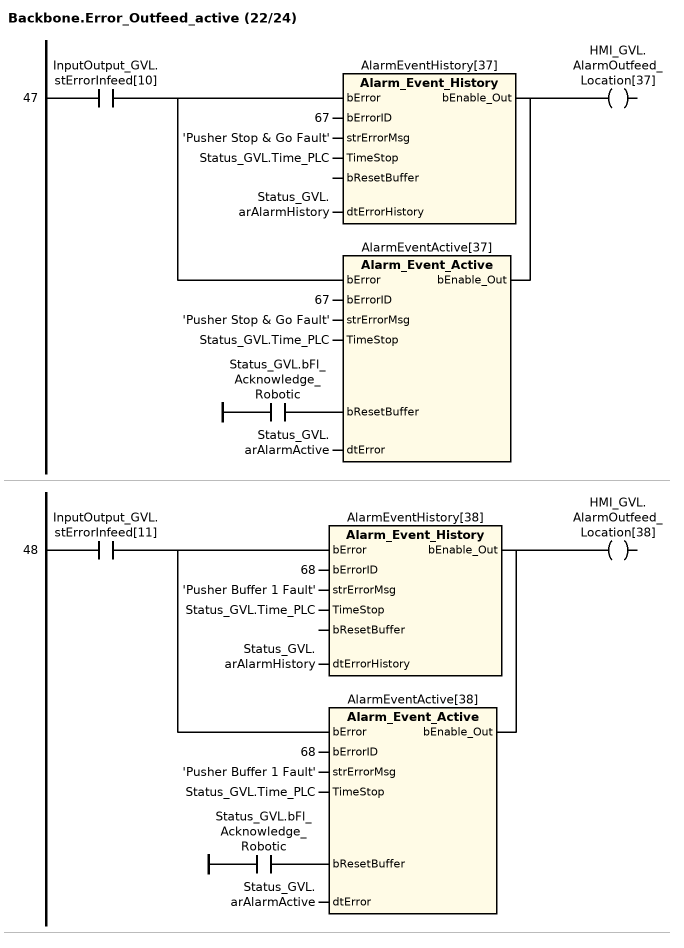
// NETWORK 47
AlarmEventHistory[37](
    bError := InputOutput_GVL.stErrorInfeed[10],
    bErrorID := 67,
    strErrorMsg := 'Pusher Stop & Go Fault',
    TimeStop := Status_GVL.Time_PLC,
    dtErrorHistory := Status_GVL.arAlarmHistory); // Alarm_Event_History
AlarmEventActive[37](
    bError := InputOutput_GVL.stErrorInfeed[10],
    bErrorID := 67,
    strErrorMsg := 'Pusher Stop & Go Fault',
    TimeStop := Status_GVL.Time_PLC,
    bResetBuffer := Status_GVL.bFl_Acknowledge_Robotic,
    dtError := Status_GVL.arAlarmActive); // Alarm_Event_Active
HMI_GVL.AlarmOutfeed_Location[37] := AlarmEventHistory[37].bEnable_Out OR AlarmEventActive[37].bEnable_Out;

// NETWORK 48
AlarmEventHistory[38](
    bError := InputOutput_GVL.stErrorInfeed[11],
    bErrorID := 68,
    strErrorMsg := 'Pusher Buffer 1 Fault',
    TimeStop := Status_GVL.Time_PLC,
    dtErrorHistory := Status_GVL.arAlarmHistory); // Alarm_Event_History
AlarmEventActive[38](
    bError := InputOutput_GVL.stErrorInfeed[11],
    bErrorID := 68,
    strErrorMsg := 'Pusher Buffer 1 Fault',
    TimeStop := Status_GVL.Time_PLC,
    bResetBuffer := Status_GVL.bFl_Acknowledge_Robotic,
    dtError := Status_GVL.arAlarmActive); // Alarm_Event_Active
HMI_GVL.AlarmOutfeed_Location[38] := AlarmEventHistory[38].bEnable_Out OR AlarmEventActive[38].bEnable_Out;

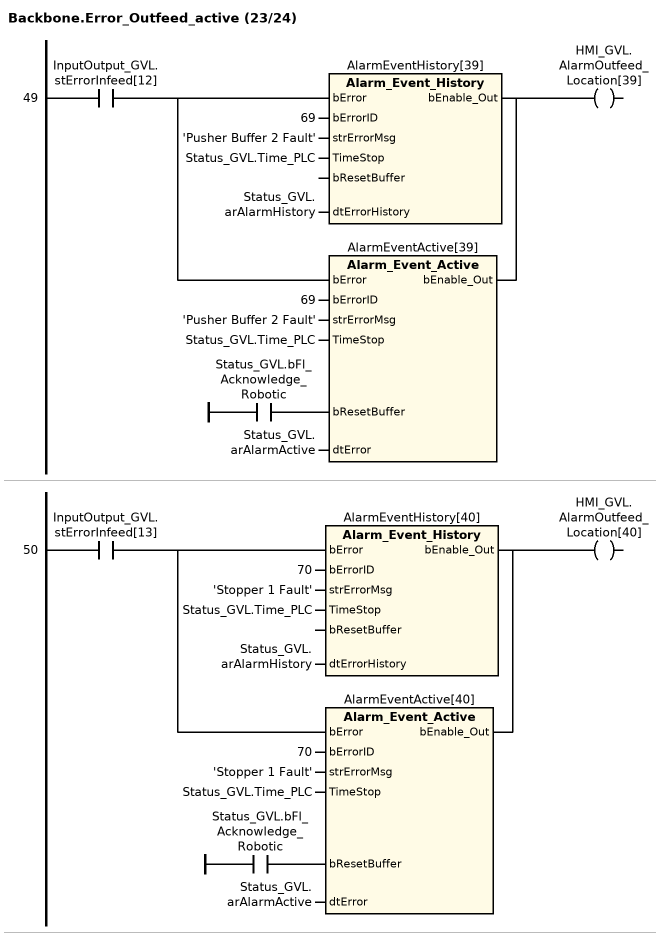
// NETWORK 49
AlarmEventHistory[39](
    bError := InputOutput_GVL.stErrorInfeed[12],
    bErrorID := 69,
    strErrorMsg := 'Pusher Buffer 2 Fault',
    TimeStop := Status_GVL.Time_PLC,
    dtErrorHistory := Status_GVL.arAlarmHistory); // Alarm_Event_History
AlarmEventActive[39](
    bError := InputOutput_GVL.stErrorInfeed[12],
    bErrorID := 69,
    strErrorMsg := 'Pusher Buffer 2 Fault',
    TimeStop := Status_GVL.Time_PLC,
    bResetBuffer := Status_GVL.bFl_Acknowledge_Robotic,
    dtError := Status_GVL.arAlarmActive); // Alarm_Event_Active
HMI_GVL.AlarmOutfeed_Location[39] := AlarmEventHistory[39].bEnable_Out OR AlarmEventActive[39].bEnable_Out;

// NETWORK 50
AlarmEventHistory[40](
    bError := InputOutput_GVL.stErrorInfeed[13],
    bErrorID := 70,
    strErrorMsg := 'Stopper 1 Fault',
    TimeStop := Status_GVL.Time_PLC,
    dtErrorHistory := Status_GVL.arAlarmHistory); // Alarm_Event_History
AlarmEventActive[40](
    bError := InputOutput_GVL.stErrorInfeed[13],
    bErrorID := 70,
    strErrorMsg := 'Stopper 1 Fault',
    TimeStop := Status_GVL.Time_PLC,
    bResetBuffer := Status_GVL.bFl_Acknowledge_Robotic,
    dtError := Status_GVL.arAlarmActive); // Alarm_Event_Active
HMI_GVL.AlarmOutfeed_Location[40] := AlarmEventHistory[40].bEnable_Out OR AlarmEventActive[40].bEnable_Out;

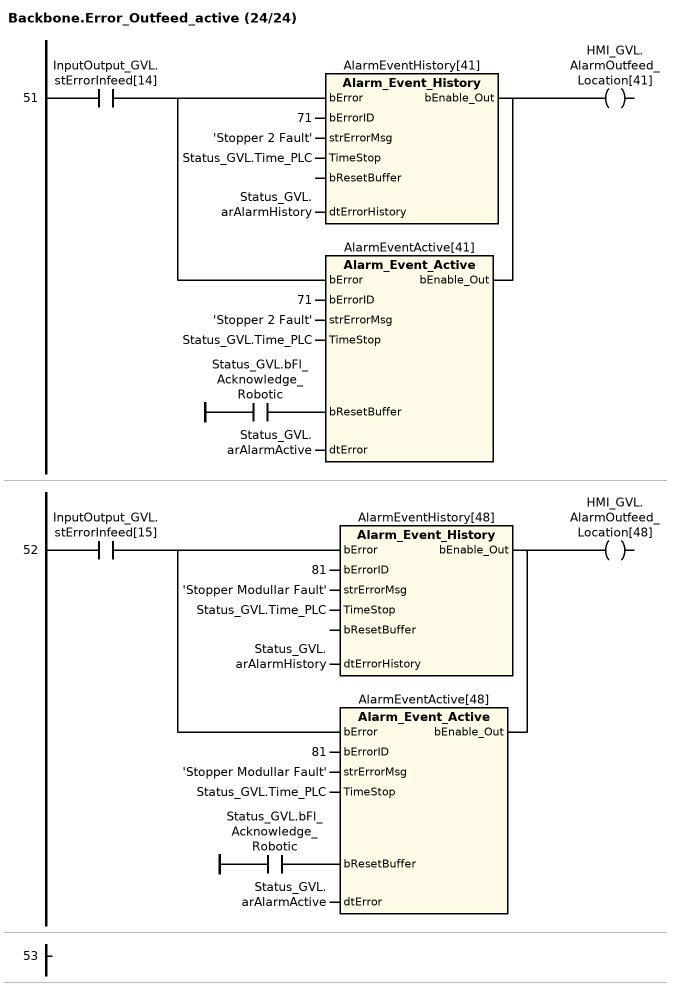
// NETWORK 51
AlarmEventHistory[41](
    bError := InputOutput_GVL.stErrorInfeed[14],
    bErrorID := 71,
    strErrorMsg := 'Stopper 2 Fault',
    TimeStop := Status_GVL.Time_PLC,
    dtErrorHistory := Status_GVL.arAlarmHistory); // Alarm_Event_History
AlarmEventActive[41](
    bError := InputOutput_GVL.stErrorInfeed[14],
    bErrorID := 71,
    strErrorMsg := 'Stopper 2 Fault',
    TimeStop := Status_GVL.Time_PLC,
    bResetBuffer := Status_GVL.bFl_Acknowledge_Robotic,
    dtError := Status_GVL.arAlarmActive); // Alarm_Event_Active
HMI_GVL.AlarmOutfeed_Location[41] := AlarmEventHistory[41].bEnable_Out OR AlarmEventActive[41].bEnable_Out;

// NETWORK 52
AlarmEventHistory[48](
    bError := InputOutput_GVL.stErrorInfeed[15],
    bErrorID := 81,
    strErrorMsg := 'Stopper Modullar Fault',
    TimeStop := Status_GVL.Time_PLC,
    dtErrorHistory := Status_GVL.arAlarmHistory); // Alarm_Event_History
AlarmEventActive[48](
    bError := InputOutput_GVL.stErrorInfeed[15],
    bErrorID := 81,
    strErrorMsg := 'Stopper Modullar Fault',
    TimeStop := Status_GVL.Time_PLC,
    bResetBuffer := Status_GVL.bFl_Acknowledge_Robotic,
    dtError := Status_GVL.arAlarmActive); // Alarm_Event_Active
HMI_GVL.AlarmOutfeed_Location[48] := AlarmEventHistory[48].bEnable_Out OR AlarmEventActive[48].bEnable_Out;

// NETWORK 53
END_ACTION

ACTION FGHS_DataCollect_active:
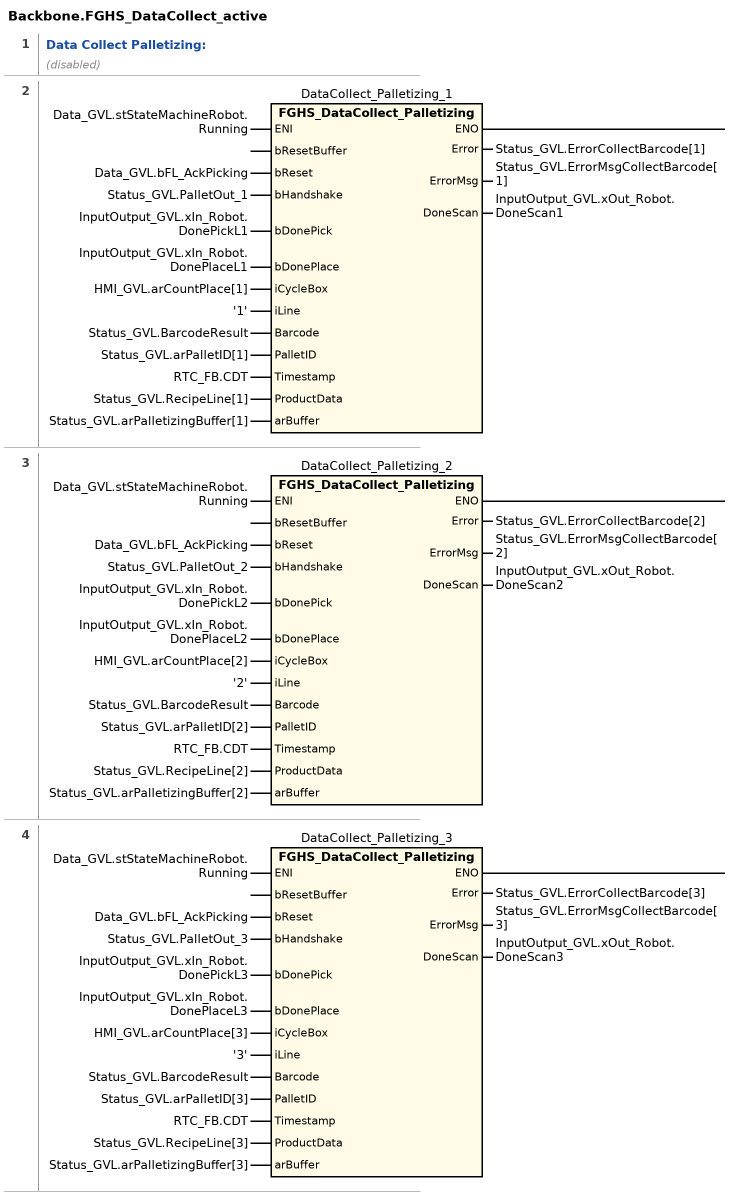
// NETWORK 1 (disabled)
// label: Data Collect Palletizing

// NETWORK 2
DataCollect_Palletizing_1(
    ENI := Data_GVL.stStateMachineRobot.Running,
    bReset := Data_GVL.bFL_AckPicking,
    bHandshake := Status_GVL.PalletOut_1,
    bDonePick := InputOutput_GVL.xIn_Robot.DonePickL1,
    bDonePlace := InputOutput_GVL.xIn_Robot.DonePlaceL1,
    iCycleBox := HMI_GVL.arCountPlace[1],
    iLine := '1',
    Barcode := Status_GVL.BarcodeResult,
    PalletID := Status_GVL.arPalletID[1],
    Timestamp := RTC_FB.CDT,
    ProductData := Status_GVL.RecipeLine[1],
    arBuffer := Status_GVL.arPalletizingBuffer[1],
    Error => Status_GVL.ErrorCollectBarcode[1],
    ErrorMsg => Status_GVL.ErrorMsgCollectBarcode[1],
    DoneScan => InputOutput_GVL.xOut_Robot.DoneScan1); // FGHS_DataCollect_Palletizing

// NETWORK 3
DataCollect_Palletizing_2(
    ENI := Data_GVL.stStateMachineRobot.Running,
    bReset := Data_GVL.bFL_AckPicking,
    bHandshake := Status_GVL.PalletOut_2,
    bDonePick := InputOutput_GVL.xIn_Robot.DonePickL2,
    bDonePlace := InputOutput_GVL.xIn_Robot.DonePlaceL2,
    iCycleBox := HMI_GVL.arCountPlace[2],
    iLine := '2',
    Barcode := Status_GVL.BarcodeResult,
    PalletID := Status_GVL.arPalletID[2],
    Timestamp := RTC_FB.CDT,
    ProductData := Status_GVL.RecipeLine[2],
    arBuffer := Status_GVL.arPalletizingBuffer[2],
    Error => Status_GVL.ErrorCollectBarcode[2],
    ErrorMsg => Status_GVL.ErrorMsgCollectBarcode[2],
    DoneScan => InputOutput_GVL.xOut_Robot.DoneScan2); // FGHS_DataCollect_Palletizing

// NETWORK 4
DataCollect_Palletizing_3(
    ENI := Data_GVL.stStateMachineRobot.Running,
    bReset := Data_GVL.bFL_AckPicking,
    bHandshake := Status_GVL.PalletOut_3,
    bDonePick := InputOutput_GVL.xIn_Robot.DonePickL3,
    bDonePlace := InputOutput_GVL.xIn_Robot.DonePlaceL3,
    iCycleBox := HMI_GVL.arCountPlace[3],
    iLine := '3',
    Barcode := Status_GVL.BarcodeResult,
    PalletID := Status_GVL.arPalletID[3],
    Timestamp := RTC_FB.CDT,
    ProductData := Status_GVL.RecipeLine[3],
    arBuffer := Status_GVL.arPalletizingBuffer[3],
    Error => Status_GVL.ErrorCollectBarcode[3],
    ErrorMsg => Status_GVL.ErrorMsgCollectBarcode[3],
    DoneScan => InputOutput_GVL.xOut_Robot.DoneScan3); // FGHS_DataCollect_Palletizing

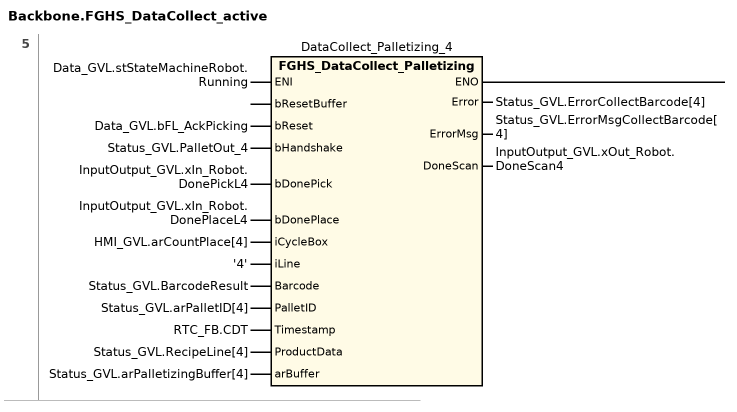
// NETWORK 5
DataCollect_Palletizing_4(
    ENI := Data_GVL.stStateMachineRobot.Running,
    bReset := Data_GVL.bFL_AckPicking,
    bHandshake := Status_GVL.PalletOut_4,
    bDonePick := InputOutput_GVL.xIn_Robot.DonePickL4,
    bDonePlace := InputOutput_GVL.xIn_Robot.DonePlaceL4,
    iCycleBox := HMI_GVL.arCountPlace[4],
    iLine := '4',
    Barcode := Status_GVL.BarcodeResult,
    PalletID := Status_GVL.arPalletID[4],
    Timestamp := RTC_FB.CDT,
    ProductData := Status_GVL.RecipeLine[4],
    arBuffer := Status_GVL.arPalletizingBuffer[4],
    Error => Status_GVL.ErrorCollectBarcode[4],
    ErrorMsg => Status_GVL.ErrorMsgCollectBarcode[4],
    DoneScan => InputOutput_GVL.xOut_Robot.DoneScan4); // FGHS_DataCollect_Palletizing
END_ACTION

ACTION FGHS_DataTraffict_active:
(* ============= Barcode Product ================= *)
//Line 1
	IF HMI_GVL.arCountReal[1] <> CheckCounter[1] THEN
		FOR Index[1] := 1 TO 60 BY 1 DO
		Status_GVL.arBarcodePallet[1,Index[1]]			:= Status_GVL.arPalletizingBuffer[1].BarcodeProduct[Index[1]];
		Status_GVL.arBarcodePalletTime[1,Index[1]]		:= Status_GVL.arPalletizingBuffer[1].BarcodeProductTime[Index[1]];
		Status_GVL.arDataPallet1[Index[1]].BarcodePallet	:= Status_GVL.arBarcodePallet[1,Index[1]];
		Status_GVL.arDataPallet1[Index[1]].BarcodePalletTime:= Status_GVL.arBarcodePalletTime[1,Index[1]]; 
		END_FOR
		CheckCounter[1]	:= HMI_GVL.arCountReal[1];
	END_IF
	
//Line 2
	IF HMI_GVL.arCountReal[2] <> CheckCounter[2] THEN
		FOR Index[2] := 1 TO 60 BY 1 DO
		Status_GVL.arBarcodePallet[2,Index[2]]			:= Status_GVL.arPalletizingBuffer[2].BarcodeProduct[Index[2]];
		Status_GVL.arBarcodePalletTime[2,Index[2]]		:= Status_GVL.arPalletizingBuffer[2].BarcodeProductTime[Index[2]];
		Status_GVL.arDataPallet2[Index[2]].BarcodePallet	:= Status_GVL.arBarcodePallet[2,Index[2]];
		Status_GVL.arDataPallet2[Index[2]].BarcodePalletTime:= Status_GVL.arBarcodePalletTime[2,Index[2]]; 
		END_FOR
		CheckCounter[2]	:= HMI_GVL.arCountReal[2];
	END_IF
	
//Line 3
	IF HMI_GVL.arCountReal[3] <> CheckCounter[3] THEN
		FOR Index[3] := 1 TO 60 BY 1 DO
		Status_GVL.arBarcodePallet[3,Index[3]]			:= Status_GVL.arPalletizingBuffer[3].BarcodeProduct[Index[3]];
		Status_GVL.arBarcodePalletTime[3,Index[3]]		:= Status_GVL.arPalletizingBuffer[3].BarcodeProductTime[Index[3]];
		Status_GVL.arDataPallet3[Index[3]].BarcodePallet	:= Status_GVL.arBarcodePallet[3,Index[3]];
		Status_GVL.arDataPallet3[Index[3]].BarcodePalletTime:= Status_GVL.arBarcodePalletTime[3,Index[3]]; 
		END_FOR
		CheckCounter[3]	:= HMI_GVL.arCountReal[3];
	END_IF
	
//Line 4
	IF HMI_GVL.arCountReal[4] <> CheckCounter[4] THEN
		FOR Index[4] := 1 TO 60 BY 1 DO
		Status_GVL.arBarcodePallet[4,Index[4]]			:= Status_GVL.arPalletizingBuffer[4].BarcodeProduct[Index[4]];
		Status_GVL.arBarcodePalletTime[4,Index[4]]		:= Status_GVL.arPalletizingBuffer[4].BarcodeProductTime[Index[4]];
		Status_GVL.arDataPallet4[Index[4]].BarcodePallet	:= Status_GVL.arBarcodePallet[4,Index[4]];
		Status_GVL.arDataPallet4[Index[4]].BarcodePalletTime:= Status_GVL.arBarcodePalletTime[4,Index[4]]; 
		END_FOR
		CheckCounter[4]	:= HMI_GVL.arCountReal[4];
	END_IF
	
	
(* ============= Link Up ================= *)
Status_GVl.arPallet_LinkUp[1]	:= Status_GVL.RecipeLine[1].LinkUpSource;
Status_GVl.arPallet_LinkUp[2]	:= Status_GVL.RecipeLine[2].LinkUpSource;
Status_GVl.arPallet_LinkUp[3]	:= Status_GVL.RecipeLine[3].LinkUpSource;
Status_GVl.arPallet_LinkUp[4]	:= Status_GVL.RecipeLine[4].LinkUpSource;


(* ============= EAN Variant ================= *)
Status_GVL.arCurrent_EAN[1]		:= Status_GVL.RecipeLine[1].EANVariant;
Status_GVL.arCurrent_EAN[2]		:= Status_GVL.RecipeLine[2].EANVariant;
Status_GVL.arCurrent_EAN[3]		:= Status_GVL.RecipeLine[3].EANVariant;
Status_GVL.arCurrent_EAN[4]		:= Status_GVL.RecipeLine[4].EANVariant;

(* ============= Code Variant ================= *)
Status_GVL.arCurrent_CodeVariant[1]		:= Status_GVL.RecipeLine[1].CodeVariant;
Status_GVL.arCurrent_CodeVariant[2]		:= Status_GVL.RecipeLine[2].CodeVariant;
Status_GVL.arCurrent_CodeVariant[3]		:= Status_GVL.RecipeLine[3].CodeVariant;
Status_GVL.arCurrent_CodeVariant[4]		:= Status_GVL.RecipeLine[4].CodeVariant;

(* ============= Interlock Infeed ================= *)
Status_GVL.ModullarInfeedBusy	:= InputOutput_GVL.Digital_Output[45];
END_ACTION

ACTION Indicator_active:
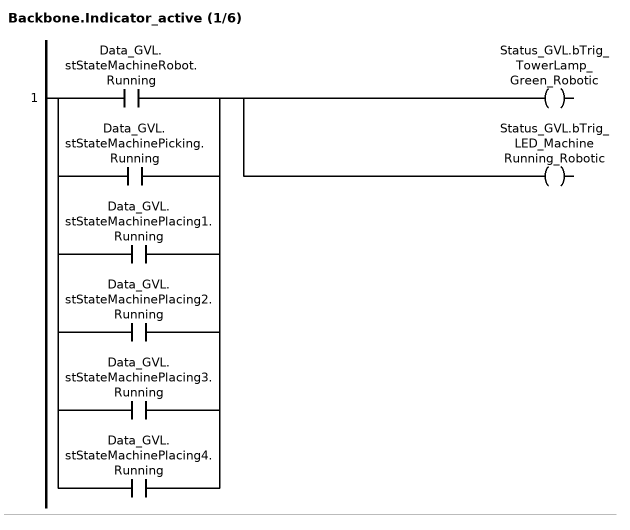
// NETWORK 1
_w1 := Data_GVL.stStateMachineRobot.Running OR Data_GVL.stStateMachinePicking.Running OR Data_GVL.stStateMachinePlacing1.Running OR Data_GVL.stStateMachinePlacing2.Running OR Data_GVL.stStateMachinePlacing3.Running OR Data_GVL.stStateMachinePlacing4.Running;
Status_GVL.bTrig_TowerLamp_Green_Robotic := _w1;
Status_GVL.bTrig_LED_MachineRunning_Robotic := _w1;

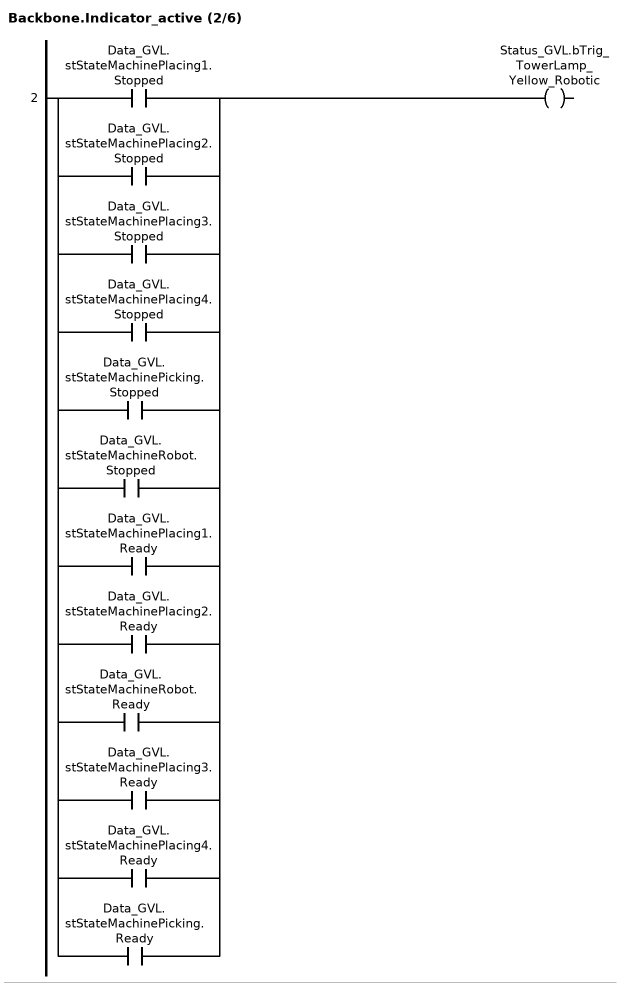
// NETWORK 2
Status_GVL.bTrig_TowerLamp_Yellow_Robotic := Data_GVL.stStateMachinePlacing1.Stopped OR Data_GVL.stStateMachinePlacing2.Stopped OR Data_GVL.stStateMachinePlacing3.Stopped OR Data_GVL.stStateMachinePlacing4.Stopped OR Data_GVL.stStateMachinePicking.Stopped OR Data_GVL.stStateMachineRobot.Stopped OR Data_GVL.stStateMachinePlacing1.Ready OR Data_GVL.stStateMachinePlacing2.Ready OR Data_GVL.stStateMachineRobot.Ready OR Data_GVL.stStateMachinePlacing3.Ready OR Data_GVL.stStateMachinePlacing4.Ready OR Data_GVL.stStateMachinePicking.Ready;

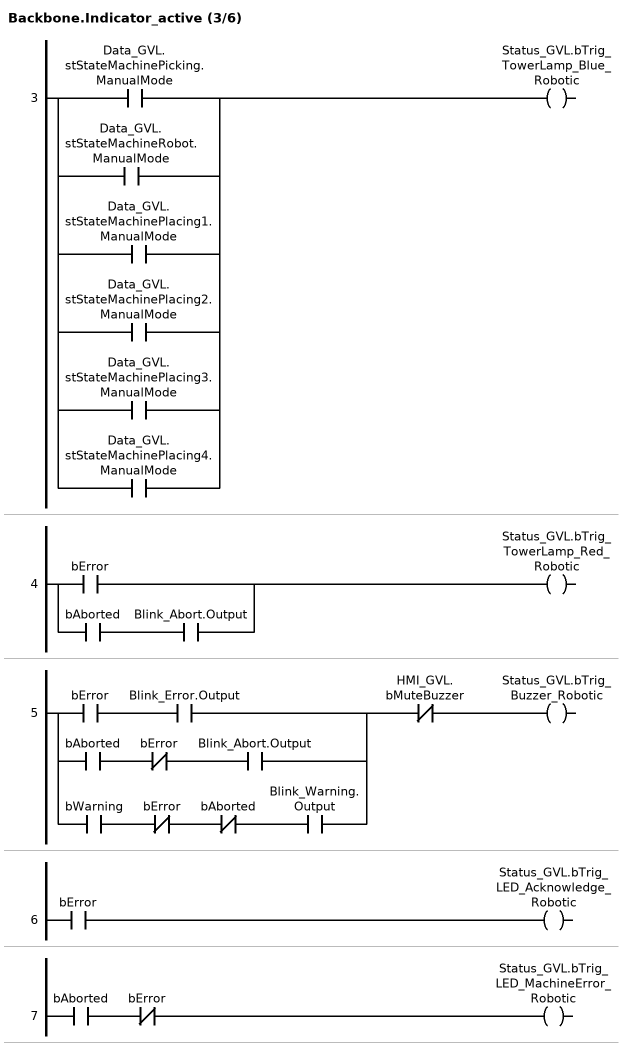
// NETWORK 3
Status_GVL.bTrig_TowerLamp_Blue_Robotic := Data_GVL.stStateMachinePicking.ManualMode OR Data_GVL.stStateMachineRobot.ManualMode OR Data_GVL.stStateMachinePlacing1.ManualMode OR Data_GVL.stStateMachinePlacing2.ManualMode OR Data_GVL.stStateMachinePlacing3.ManualMode OR Data_GVL.stStateMachinePlacing4.ManualMode;

// NETWORK 4
Status_GVL.bTrig_TowerLamp_Red_Robotic := bError OR bAborted AND Blink_Abort.Output;

// NETWORK 5
Status_GVL.bTrig_Buzzer_Robotic := (bError AND Blink_Error.Output OR bAborted AND NOT bError AND Blink_Abort.Output OR bWarning AND NOT bError AND NOT bAborted AND Blink_Warning.Output) AND NOT HMI_GVL.bMuteBuzzer;

// NETWORK 6
Status_GVL.bTrig_LED_Acknowledge_Robotic := bError;

// NETWORK 7
Status_GVL.bTrig_LED_MachineError_Robotic := bAborted AND NOT bError;

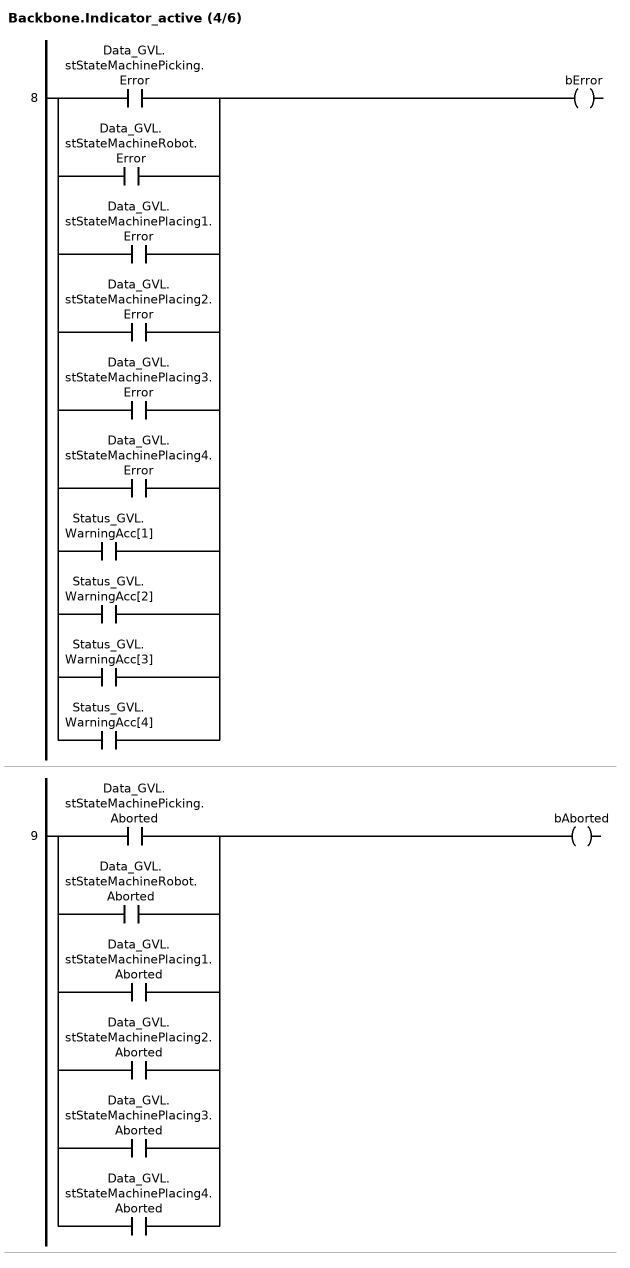
// NETWORK 8
bError := Data_GVL.stStateMachinePicking.Error OR Data_GVL.stStateMachineRobot.Error OR Data_GVL.stStateMachinePlacing1.Error OR Data_GVL.stStateMachinePlacing2.Error OR Data_GVL.stStateMachinePlacing3.Error OR Data_GVL.stStateMachinePlacing4.Error OR Status_GVL.WarningAcc[1] OR Status_GVL.WarningAcc[2] OR Status_GVL.WarningAcc[3] OR Status_GVL.WarningAcc[4];

// NETWORK 9
bAborted := Data_GVL.stStateMachinePicking.Aborted OR Data_GVL.stStateMachineRobot.Aborted OR Data_GVL.stStateMachinePlacing1.Aborted OR Data_GVL.stStateMachinePlacing2.Aborted OR Data_GVL.stStateMachinePlacing3.Aborted OR Data_GVL.stStateMachinePlacing4.Aborted;

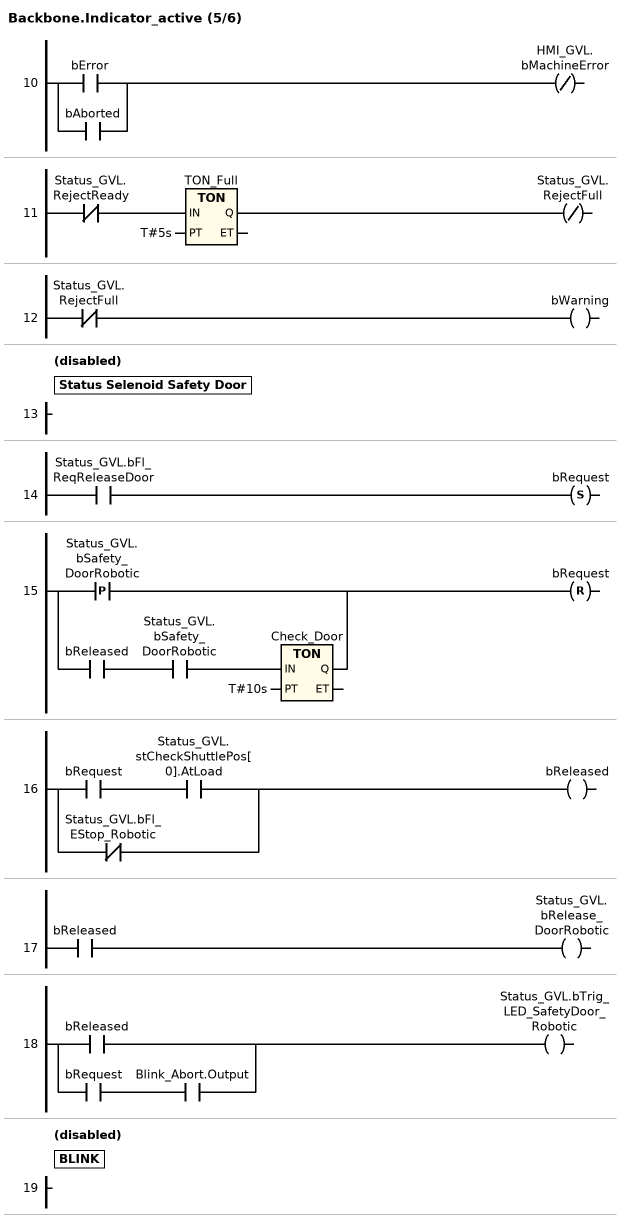
// NETWORK 10
HMI_GVL.bMachineError := NOT (bError OR bAborted);

// NETWORK 11
TON_Full(IN := NOT Status_GVL.RejectReady, PT := T#5s); // TON
Status_GVL.RejectFull := NOT TON_Full.Q;

// NETWORK 12
bWarning := NOT Status_GVL.RejectFull;

// NETWORK 13 (disabled)
// label: Status Selenoid Safety Door

// NETWORK 14
bRequest S= Status_GVL.bFl_ReqReleaseDoor;

// NETWORK 15
_rt1(CLK := Status_GVL.bSafety_DoorRobotic);
Check_Door(IN := bReleased AND Status_GVL.bSafety_DoorRobotic, PT := T#10s); // TON
bRequest R= _rt1.Q OR Check_Door.Q;

// NETWORK 16
bReleased := bRequest AND Status_GVL.stCheckShuttlePos[0].AtLoad OR NOT Status_GVL.bFl_EStop_Robotic;

// NETWORK 17
Status_GVL.bRelease_DoorRobotic := bReleased;

// NETWORK 18
Status_GVL.bTrig_LED_SafetyDoor_Robotic := bReleased OR bRequest AND Blink_Abort.Output;

// NETWORK 19 (disabled)
// label: BLINK

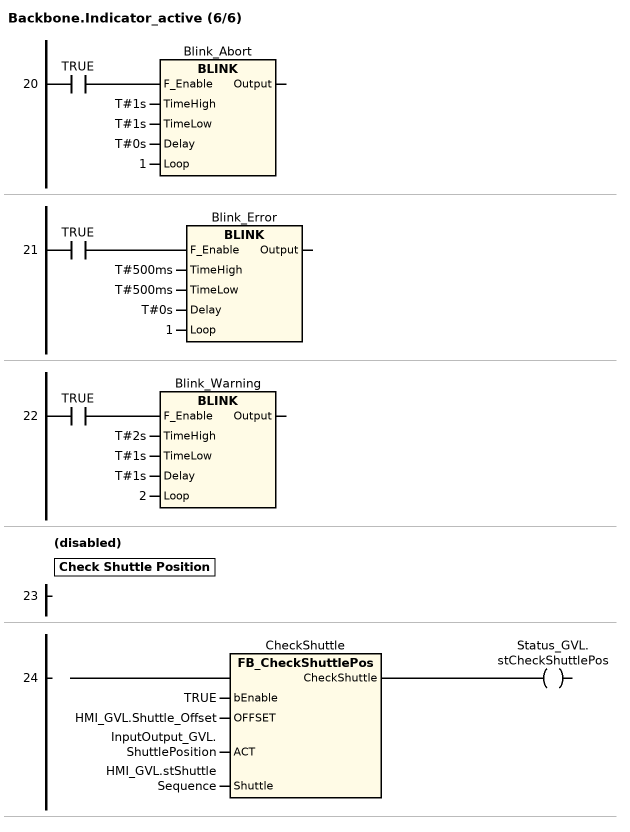
// NETWORK 20
Blink_Abort(F_Enable := TRUE, TimeHigh := T#1s, TimeLow := T#1s, Delay := T#0s, Loop := 1); // BLINK

// NETWORK 21
Blink_Error(F_Enable := TRUE, TimeHigh := T#500ms, TimeLow := T#500ms, Delay := T#0s, Loop := 1); // BLINK

// NETWORK 22
Blink_Warning(F_Enable := TRUE, TimeHigh := T#2s, TimeLow := T#1s, Delay := T#1s, Loop := 2); // BLINK

// NETWORK 23 (disabled)
// label: Check Shuttle Position

// NETWORK 24
CheckShuttle(
    bEnable := TRUE,
    OFFSET := HMI_GVL.Shuttle_Offset,
    ACT := InputOutput_GVL.ShuttlePosition,
    Shuttle := HMI_GVL.stShuttleSequence); // FB_CheckShuttlePos
Status_GVL.stCheckShuttlePos := CheckShuttle.CheckShuttle;
END_ACTION

ACTION OEE_active:
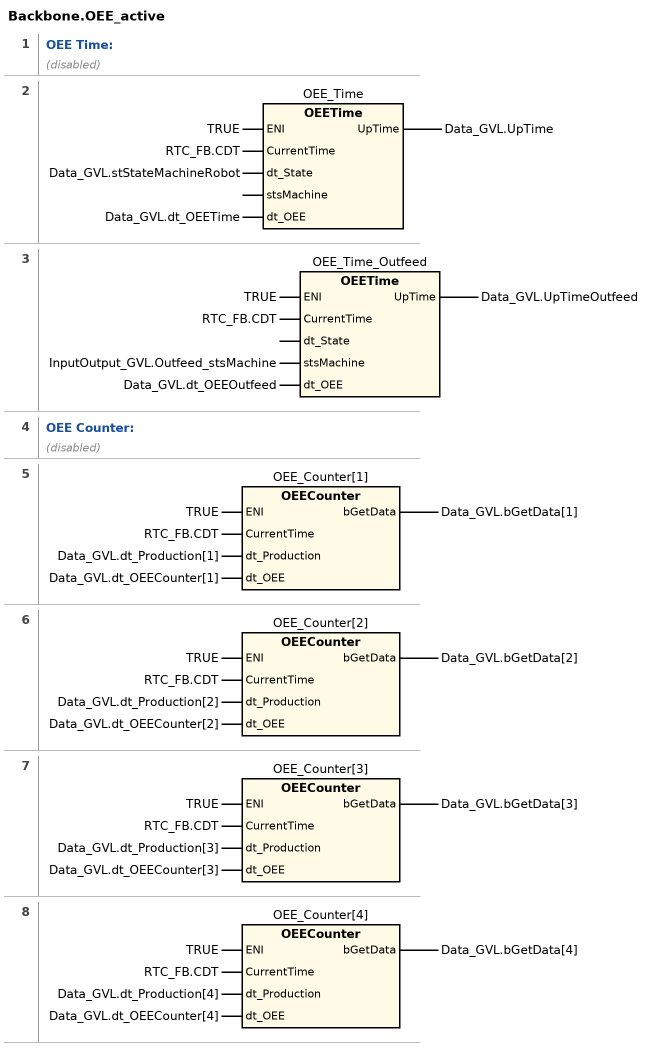
// NETWORK 1 (disabled)
// label: OEE Time

// NETWORK 2
OEE_Time(
    ENI := TRUE,
    CurrentTime := RTC_FB.CDT,
    dt_State := Data_GVL.stStateMachineRobot,
    dt_OEE := Data_GVL.dt_OEETime); // OEETime
Data_GVL.UpTime := OEE_Time.UpTime;

// NETWORK 3
OEE_Time_Outfeed(
    ENI := TRUE,
    CurrentTime := RTC_FB.CDT,
    stsMachine := InputOutput_GVL.Outfeed_stsMachine,
    dt_OEE := Data_GVL.dt_OEEOutfeed); // OEETime
Data_GVL.UpTimeOutfeed := OEE_Time_Outfeed.UpTime;

// NETWORK 4 (disabled)
// label: OEE Counter

// NETWORK 5
OEE_Counter[1](
    ENI := TRUE,
    CurrentTime := RTC_FB.CDT,
    dt_Production := Data_GVL.dt_Production[1],
    dt_OEE := Data_GVL.dt_OEECounter[1]); // OEECounter
Data_GVL.bGetData[1] := OEE_Counter[1].bGetData;

// NETWORK 6
OEE_Counter[2](
    ENI := TRUE,
    CurrentTime := RTC_FB.CDT,
    dt_Production := Data_GVL.dt_Production[2],
    dt_OEE := Data_GVL.dt_OEECounter[2]); // OEECounter
Data_GVL.bGetData[2] := OEE_Counter[2].bGetData;

// NETWORK 7
OEE_Counter[3](
    ENI := TRUE,
    CurrentTime := RTC_FB.CDT,
    dt_Production := Data_GVL.dt_Production[3],
    dt_OEE := Data_GVL.dt_OEECounter[3]); // OEECounter
Data_GVL.bGetData[3] := OEE_Counter[3].bGetData;

// NETWORK 8
OEE_Counter[4](
    ENI := TRUE,
    CurrentTime := RTC_FB.CDT,
    dt_Production := Data_GVL.dt_Production[4],
    dt_OEE := Data_GVL.dt_OEECounter[4]); // OEECounter
Data_GVL.bGetData[4] := OEE_Counter[4].bGetData;
END_ACTION

ACTION Parameter_Outfeed_active:
//Safety Outfeed
InputOutput_GVL.TestMode[99]	:= NOT Status_GVL.bFl_EStop_Robotic OR NOT Status_GVL.bSafety_DoorRobotic OR Backbone.bRequest;

//Mute Buzzer
InputOutput_GVL.TestMode[98]	:= HMI_GVL.bMuteBuzzer;

//Disable Overflow
InputOutput_GVL.TestMode[97]	:= HMI_GVL.Disable_Overflow;

//Lock Modullar to Keep Running
InputOutput_GVL.TestMode[96]	:= HMI_GVL.LockModullarToRun;

//Ack Button Outfeed
InputOutput_GVL.TestMode[95]	:= Status_GVL.bFl_Acknowledge_Robotic;

//Reset Button Outfeed
InputOutput_GVL.TestMode[94]	:= Status_GVL.bFl_ResetButton_Robotic;

//Status Running Picking
InputOutput_GVL.TestMode[93]	:= Data_GVL.stStateMachinePicking.Running;

//Bypass Wrapper
InputOutput_GVL.TestMode[92]	:= HMI_GVL.BypassWrapper;

//Bypass Wrapper Existing
InputOutput_GVL.TestMode[91]	:= HMI_GVL.BypassWrapperExisting;

(*================= Control Button ============================*) 
InputOutput_GVL.ControlButton[1]					:= HMI_GVL.bStartButtonOutfeed;
InputOutput_GVL.ControlButton[2]					:= HMI_GVL.bStopButtonOutfeed;
InputOutput_GVL.ControlButton[3]					:= HMI_GVL.bResetButtonOutfeed;
InputOutput_GVL.ControlButton[4]					:= HMI_GVL.bTestModeEnableOutfeed;
InputOutput_GVL.ControlButton[5]					:= HMI_GVL.bAcknowledgeButtonOutfeed;

InputOutput_GVL.ControlButton[6]					:= HMI_GVL.bStartButtonShuttle;
InputOutput_GVL.ControlButton[7]					:= HMI_GVL.bStopButtonShuttle;
InputOutput_GVL.ControlButton[8]					:= HMI_GVL.bResetButtonShuttle;
InputOutput_GVL.ControlButton[9]					:= HMI_GVL.bTestModeEnableShuttle;
InputOutput_GVL.ControlButton[10]					:= HMI_GVL.bAcknowledgeButtonShuttle;

InputOutput_GVL.ControlButton[11]					:= HMI_GVL.bStartButtonDispenser;
InputOutput_GVL.ControlButton[12]					:= HMI_GVL.bStopButtonDispenser;
InputOutput_GVL.ControlButton[13]					:= HMI_GVL.bResetButtonDispenser;
InputOutput_GVL.ControlButton[14]					:= HMI_GVL.bTestModeEnableDispenser;
InputOutput_GVL.ControlButton[15]					:= HMI_GVL.bAcknowledgeButtonDispenser;

InputOutput_GVL.ControlButton[16]					:= HMI_GVL.bStartButtonInfeed;
InputOutput_GVL.ControlButton[17]					:= HMI_GVL.bStopButtonInfeed;
InputOutput_GVL.ControlButton[18]					:= HMI_GVL.bResetButtonInfeed;
InputOutput_GVL.ControlButton[19]					:= HMI_GVL.bTestModeEnableInfeed;
InputOutput_GVL.ControlButton[20]					:= HMI_GVL.bAcknowledgeButtonInfeed;


(*================= Parameter Shuttle ============================*)
//Handshake Shuttle
InputOutput_GVL.RequestEmptyPallet[1]	:= Status_GVL.RequestEmptyPallet[1];
InputOutput_GVL.RequestEmptyPallet[2]	:= Status_GVL.RequestEmptyPallet[2];
InputOutput_GVL.RequestEmptyPallet[3]	:= Status_GVL.RequestEmptyPallet[3];
InputOutput_GVL.RequestEmptyPallet[4]	:= Status_GVL.RequestEmptyPallet[4];

InputOutput_GVL.RequestLoadPallet[1]	:= Status_GVL.RequestLoadPallet[1];
InputOutput_GVL.RequestLoadPallet[2]	:= Status_GVL.RequestLoadPallet[2];
InputOutput_GVL.RequestLoadPallet[3]	:= Status_GVL.RequestLoadPallet[3];
InputOutput_GVL.RequestLoadPallet[4]	:= Status_GVL.RequestLoadPallet[4];

Status_GVL.FB_RequestShuttle[1]			:= InputOutput_GVL.FB_RequestShuttle[1];
Status_GVL.FB_RequestShuttle[2]			:= InputOutput_GVL.FB_RequestShuttle[2];
Status_GVL.FB_RequestShuttle[3]			:= InputOutput_GVL.FB_RequestShuttle[3];
Status_GVL.FB_RequestShuttle[4]			:= InputOutput_GVL.FB_RequestShuttle[4];


//Shuttle Position
//InputOutput_GVL.TestMode[100] ==> Download Parameter Shuttle Position	
InputOutput_GVL.stShuttleSequence[0].PositionEmpty	:= HMI_GVL.stShuttleSequence[0].PositionEmpty;
InputOutput_GVL.stShuttleSequence[1].PositionEmpty	:= HMI_GVL.stShuttleSequence[1].PositionEmpty;
InputOutput_GVL.stShuttleSequence[2].PositionEmpty	:= HMI_GVL.stShuttleSequence[2].PositionEmpty;
InputOutput_GVL.stShuttleSequence[3].PositionEmpty	:= HMI_GVL.stShuttleSequence[3].PositionEmpty;
InputOutput_GVL.stShuttleSequence[4].PositionEmpty	:= HMI_GVL.stShuttleSequence[4].PositionEmpty;

InputOutput_GVL.stShuttleSequence[0].PositionLoaded	:= HMI_GVL.stShuttleSequence[0].PositionLoaded;
InputOutput_GVL.stShuttleSequence[1].PositionLoaded	:= HMI_GVL.stShuttleSequence[1].PositionLoaded;
InputOutput_GVL.stShuttleSequence[2].PositionLoaded	:= HMI_GVL.stShuttleSequence[2].PositionLoaded;
InputOutput_GVL.stShuttleSequence[3].PositionLoaded	:= HMI_GVL.stShuttleSequence[3].PositionLoaded;
InputOutput_GVL.stShuttleSequence[4].PositionLoaded	:= HMI_GVL.stShuttleSequence[4].PositionLoaded;

//Shuttle Speed
InputOutput_GVL.Shuttle_Speed[1]					:= HMI_GVL.Shuttle_JogSpeed;
InputOutput_GVL.Shuttle_Speed[2]					:= HMI_GVL.Shuttle_MinSpeed;
InputOutput_GVL.Shuttle_Speed[3]					:= HMI_GVL.Shuttle_MaxSpeed;
InputOutput_GVL.Shuttle_Offset						:= HMI_GVL.Shuttle_Offset;

//Counter Box at Placing
InputOutput_GVL.Counter[1]							:= HMI_GVL.arCountReal[1];
InputOutput_GVL.Counter[2]							:= HMI_GVL.arCountReal[2];
InputOutput_GVL.Counter[3]							:= HMI_GVL.arCountReal[3];
InputOutput_GVL.Counter[4]							:= HMI_GVL.arCountReal[4];


(*================= Parameter Timer ============================*)
//=====> Shuttle
InputOutput_GVL.TmrOutfeed[1]						:= HMI_GVL.Tmr_EmptyShuttle;
InputOutput_GVL.TmrOutfeed[2]						:= HMI_GVL.Tmr_LoadedShuttle;
InputOutput_GVL.TmrOutfeed[3]						:= HMI_GVL.Tmr_BrakeShuttle; 

//=====> Outfeed
InputOutput_GVL.TmrOutfeed[4]						:= HMI_GVL.Tmr_PalletBuffer2;
InputOutput_GVL.TmrOutfeed[5]						:= HMI_GVL.Tmr_PalletBuffer1;
InputOutput_GVL.TmrOutfeed[6]						:= HMI_GVL.Tmr_PalletOutfeed1;
InputOutput_GVL.TmrOutfeed[7]						:= HMI_GVL.Tmr_PalletOutfeed2;
InputOutput_GVL.TmrOutfeed[8]						:= HMI_GVL.Tmr_PalletOutfeed3;
InputOutput_GVL.TmrOutfeed[9]						:= HMI_GVL.Tmr_PalletOutfeed4;
InputOutput_GVL.TmrOutfeed[10]						:= HMI_GVL.Tmr_PalletOutfeed5;
InputOutput_GVL.TmrOutfeed[11]						:= HMI_GVL.Tmr_PalletRA;
InputOutput_GVL.TmrOutfeed[12]						:= HMI_GVL.TmrDelay_PalletRA;

//=====> Infeed
InputOutput_GVL.TmrOutfeed[13]						:= HMI_GVL.Tmr_Stopper1;
InputOutput_GVL.TmrOutfeed[14]						:= HMI_GVL.Tmr_Stopper2;
InputOutput_GVL.TmrOutfeed[15]						:= HMI_GVL.Tmr_StopGo;
InputOutput_GVL.TmrOutfeed[16]						:= HMI_GVL.Tmr_Infeed;
InputOutput_GVL.TmrOutfeed[17]						:= HMI_GVL.Tmr_Buffer1;
InputOutput_GVL.TmrOutfeed[18]						:= HMI_GVL.Tmr_Buffer2;
InputOutput_GVL.TmrOutfeed[19]						:= HMI_GVL.Tmr_ModullarOn;
InputOutput_GVL.TmrOutfeed[20]						:= HMI_GVL.Tmr_ModullarOff;

//=====> Dispenser
InputOutput_GVL.TmrOutfeed[21]						:= HMI_GVL.Tmr_Dispenser;

(*================= SeqIndex ============================*)
//Shuttle Empty
CASE InputOutput_GVL.SeqIndexOutfeed[1] OF
	0:		HMI_GVL.CJ_ShuttleEmpty	:= 'Check Sensor';
	100:	HMI_GVL.CJ_ShuttleEmpty	:= 'Request to Dispenser';
	110:	HMI_GVL.CJ_ShuttleEmpty	:= 'Empty Pallet In';
	500:	HMI_GVL.CJ_ShuttleEmpty	:= 'Empty Pallet Ready';
	600:	HMI_GVL.CJ_ShuttleEmpty	:= 'Empty Pallet Out';
END_CASE

//Shuttle Load
CASE InputOutput_GVL.SeqIndexOutfeed[2] OF
	0:		HMI_GVL.CJ_ShuttleLoad	:= 'Check Sensor';
	100:	HMI_GVL.CJ_ShuttleLoad	:= 'Waiting to Pick Up Loaded Pallet';
	101:	HMI_GVL.CJ_ShuttleLoad	:= 'Unloading Pallet In';
	110:	HMI_GVL.CJ_ShuttleLoad	:= 'Loaded Pallet In';
	500:	HMI_GVL.CJ_ShuttleLoad	:= 'Loaded Pallet Ready';
	600:	HMI_GVL.CJ_ShuttleLoad	:= 'Loaded Pallet Out';
END_CASE


//Shuttle Management
CASE InputOutput_GVL.SeqIndexOutfeed[3] OF
	0:		HMI_GVL.CJ_ShuttleManagement	:= 'Standby';
	100:	HMI_GVL.CJ_ShuttleManagement	:= 'Move to Standby';
	
	1001:	HMI_GVL.CJ_ShuttleManagement	:= 'Move to Dispenser - Outfeed';
	1020:	HMI_GVL.CJ_ShuttleManagement	:= 'Shuttle at Dispenser - Outfeed';
	1030:	HMI_GVL.CJ_ShuttleManagement	:= 'Transfer Pallet at Dispenser - Outfeed';
	1100:	HMI_GVL.CJ_ShuttleManagement	:= 'Done Transfer Pallet at Dispenser - Outfeed';
	
	2001:	HMI_GVL.CJ_ShuttleManagement	:= 'Move to Unloading';
	2020:	HMI_GVL.CJ_ShuttleManagement	:= 'Request Load Pallet from Unloading';
	2030:	HMI_GVL.CJ_ShuttleManagement	:= 'Unloading Pallet In';
	2040:	HMI_GVL.CJ_ShuttleManagement	:= 'Check Request from Outfeed';
	2050:	HMI_GVL.CJ_ShuttleManagement	:= 'Transfer Load Pallet to Outfeed';
	2100:	HMI_GVL.CJ_ShuttleManagement	:= 'Done Unloading';
	
	3000:	HMI_GVL.CJ_ShuttleManagement	:= 'Waiting for Request Line';
	3001:	HMI_GVL.CJ_ShuttleManagement	:= 'Waiting for Request Line';
	3002:	HMI_GVL.CJ_ShuttleManagement	:= 'Waiting for Request Line';
	3003:	HMI_GVL.CJ_ShuttleManagement	:= 'Waiting for Request Line';
	3004:	HMI_GVL.CJ_ShuttleManagement	:= 'Waiting for Request Line';
	3011:	HMI_GVL.CJ_ShuttleManagement	:= 'Loaded Pallet Transfer From Line 1';
	3012:	HMI_GVL.CJ_ShuttleManagement	:= 'Loaded Pallet Transfer From Line 2';
	3013:	HMI_GVL.CJ_ShuttleManagement	:= 'Loaded Pallet Transfer From Line 3';
	3014:	HMI_GVL.CJ_ShuttleManagement	:= 'Loaded Pallet Transfer From Line 4';
	3041:	HMI_GVL.CJ_ShuttleManagement	:= 'Transfer Load Pallet from Line 1';
	3042:	HMI_GVL.CJ_ShuttleManagement	:= 'Transfer Load Pallet from Line 2';
	3043:	HMI_GVL.CJ_ShuttleManagement	:= 'Transfer Load Pallet from Line 3';
	3044:	HMI_GVL.CJ_ShuttleManagement	:= 'Transfer Load Pallet from Line 4';
	3051:	HMI_GVL.CJ_ShuttleManagement	:= 'Empty Pallet Transfer To Line 1';
	3052:	HMI_GVL.CJ_ShuttleManagement	:= 'Empty Pallet Transfer To Line 2';
	3053:	HMI_GVL.CJ_ShuttleManagement	:= 'Empty Pallet Transfer To Line 3';
	3054:	HMI_GVL.CJ_ShuttleManagement	:= 'Empty Pallet Transfer To Line 4';
	3091:	HMI_GVL.CJ_ShuttleManagement	:= 'Transfer Empty Pallet to Line 1';
	3092:	HMI_GVL.CJ_ShuttleManagement	:= 'Transfer Empty Pallet to Line 2';
	3093:	HMI_GVL.CJ_ShuttleManagement	:= 'Transfer Empty Pallet to Line 3';
	3094:	HMI_GVL.CJ_ShuttleManagement	:= 'Transfer Empty Pallet to Line 4';
	3100:	HMI_GVL.CJ_ShuttleManagement	:= 'Done Standby';
	
END_CASE

//Dispenser
CASE InputOutput_GVL.SeqIndexOutfeed[4] OF
	0:		HMI_GVL.CJ_Dispenser	:= 'Check Pallet';
	10:		HMI_GVL.CJ_Dispenser	:= 'Move Pneu Vertical to Middle';
	20:		HMI_GVL.CJ_Dispenser	:= 'Check Sensor Stack';
	50:		HMI_GVL.CJ_Dispenser	:= 'Pneu Horizontal Retract';
	100:	HMI_GVL.CJ_Dispenser	:= 'Move Pneu Vertical to Bottom';
	150:	HMI_GVL.CJ_Dispenser	:= 'Request Pallet';
	200:	HMI_GVL.CJ_Dispenser	:= 'Pallet In';
	500:	HMI_GVL.CJ_Dispenser	:= 'Check Stack Pallet';
	520:	HMI_GVL.CJ_Dispenser	:= 'Pneu Horizontal Retract';
	550:	HMI_GVL.CJ_Dispenser	:= 'Move Pneu Vertical to Middle';
	555:	HMI_GVL.CJ_Dispenser	:= 'Move Pneu Vertical to Middle';
	600:	HMI_GVL.CJ_Dispenser	:= 'Pneu Horizontal Advance';
	650:	HMI_GVL.CJ_Dispenser	:= 'Move Pneu Vertical to Top';
	700:	HMI_GVL.CJ_Dispenser	:= 'Transfer Pallet Out';
	750:	HMI_GVL.CJ_Dispenser	:= 'Move Pneu Vertical to Bottom';
	800:	HMI_GVL.CJ_Dispenser	:= 'Pneu Horizontal Retract';
	
END_CASE
END_ACTION

ACTION Recipe_active:
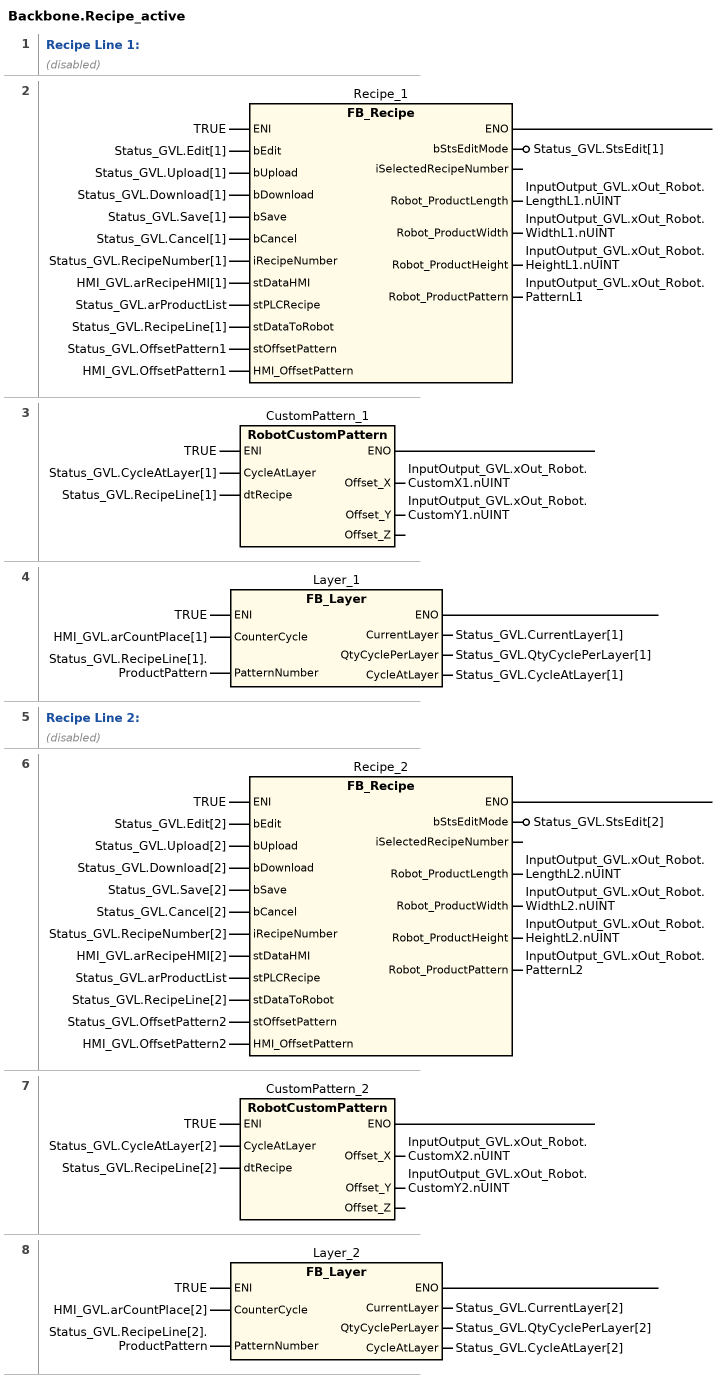
// NETWORK 1 (disabled)
// label: Recipe Line 1

// NETWORK 2
Recipe_1(
    ENI := TRUE,
    bEdit := Status_GVL.Edit[1],
    bUpload := Status_GVL.Upload[1],
    bDownload := Status_GVL.Download[1],
    bSave := Status_GVL.Save[1],
    bCancel := Status_GVL.Cancel[1],
    iRecipeNumber := Status_GVL.RecipeNumber[1],
    stDataHMI := HMI_GVL.arRecipeHMI[1],
    stPLCRecipe := Status_GVL.arProductList,
    stDataToRobot := Status_GVL.RecipeLine[1],
    stOffsetPattern := Status_GVL.OffsetPattern1,
    HMI_OffsetPattern := HMI_GVL.OffsetPattern1,
    Robot_ProductLength => InputOutput_GVL.xOut_Robot.LengthL1.nUINT,
    Robot_ProductWidth => InputOutput_GVL.xOut_Robot.WidthL1.nUINT,
    Robot_ProductHeight => InputOutput_GVL.xOut_Robot.HeightL1.nUINT,
    Robot_ProductPattern => InputOutput_GVL.xOut_Robot.PatternL1); // FB_Recipe
Status_GVL.StsEdit[1] := NOT Recipe_1.bStsEditMode;

// NETWORK 3
CustomPattern_1(
    ENI := TRUE,
    CycleAtLayer := Status_GVL.CycleAtLayer[1],
    dtRecipe := Status_GVL.RecipeLine[1],
    Offset_X => InputOutput_GVL.xOut_Robot.CustomX1.nUINT,
    Offset_Y => InputOutput_GVL.xOut_Robot.CustomY1.nUINT); // RobotCustomPattern

// NETWORK 4
Layer_1(
    ENI := TRUE,
    CounterCycle := HMI_GVL.arCountPlace[1],
    PatternNumber := Status_GVL.RecipeLine[1].ProductPattern,
    CurrentLayer => Status_GVL.CurrentLayer[1],
    QtyCyclePerLayer => Status_GVL.QtyCyclePerLayer[1],
    CycleAtLayer => Status_GVL.CycleAtLayer[1]); // FB_Layer

// NETWORK 5 (disabled)
// label: Recipe Line 2

// NETWORK 6
Recipe_2(
    ENI := TRUE,
    bEdit := Status_GVL.Edit[2],
    bUpload := Status_GVL.Upload[2],
    bDownload := Status_GVL.Download[2],
    bSave := Status_GVL.Save[2],
    bCancel := Status_GVL.Cancel[2],
    iRecipeNumber := Status_GVL.RecipeNumber[2],
    stDataHMI := HMI_GVL.arRecipeHMI[2],
    stPLCRecipe := Status_GVL.arProductList,
    stDataToRobot := Status_GVL.RecipeLine[2],
    stOffsetPattern := Status_GVL.OffsetPattern2,
    HMI_OffsetPattern := HMI_GVL.OffsetPattern2,
    Robot_ProductLength => InputOutput_GVL.xOut_Robot.LengthL2.nUINT,
    Robot_ProductWidth => InputOutput_GVL.xOut_Robot.WidthL2.nUINT,
    Robot_ProductHeight => InputOutput_GVL.xOut_Robot.HeightL2.nUINT,
    Robot_ProductPattern => InputOutput_GVL.xOut_Robot.PatternL2); // FB_Recipe
Status_GVL.StsEdit[2] := NOT Recipe_2.bStsEditMode;

// NETWORK 7
CustomPattern_2(
    ENI := TRUE,
    CycleAtLayer := Status_GVL.CycleAtLayer[2],
    dtRecipe := Status_GVL.RecipeLine[2],
    Offset_X => InputOutput_GVL.xOut_Robot.CustomX2.nUINT,
    Offset_Y => InputOutput_GVL.xOut_Robot.CustomY2.nUINT); // RobotCustomPattern

// NETWORK 8
Layer_2(
    ENI := TRUE,
    CounterCycle := HMI_GVL.arCountPlace[2],
    PatternNumber := Status_GVL.RecipeLine[2].ProductPattern,
    CurrentLayer => Status_GVL.CurrentLayer[2],
    QtyCyclePerLayer => Status_GVL.QtyCyclePerLayer[2],
    CycleAtLayer => Status_GVL.CycleAtLayer[2]); // FB_Layer

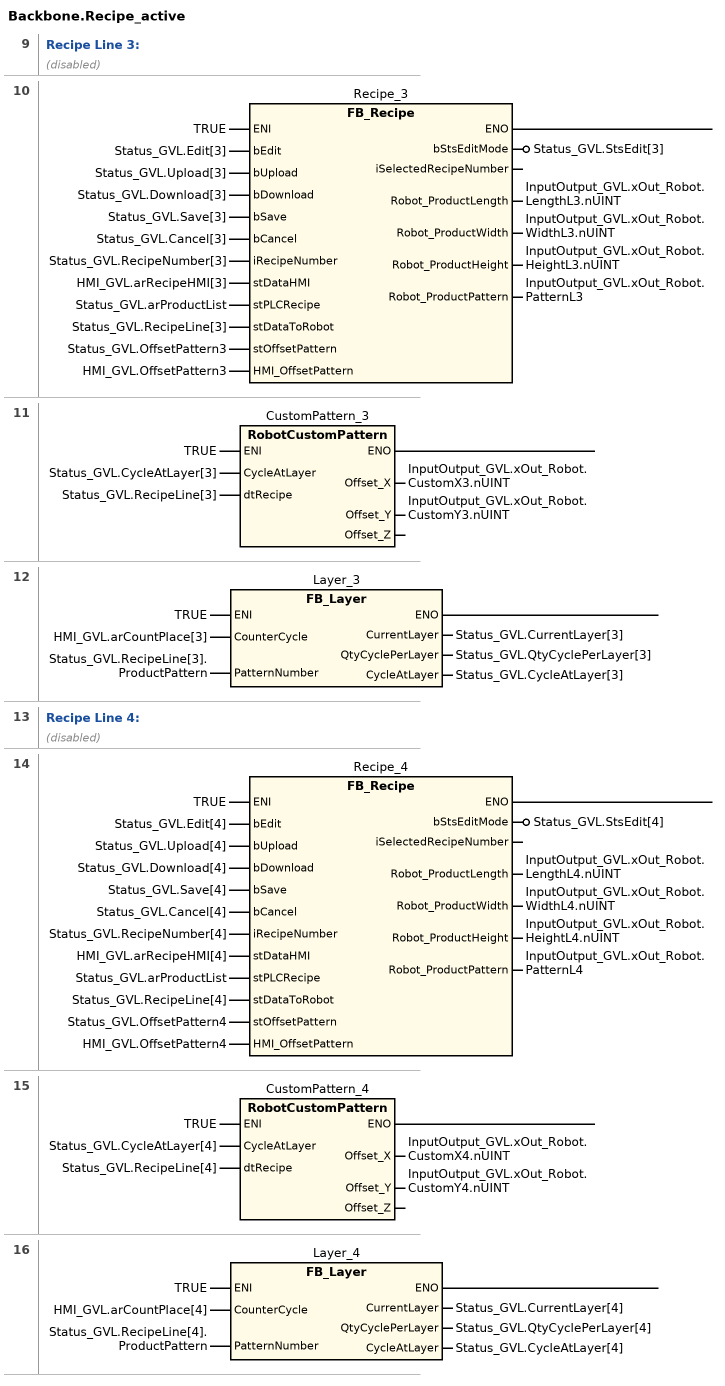
// NETWORK 9 (disabled)
// label: Recipe Line 3

// NETWORK 10
Recipe_3(
    ENI := TRUE,
    bEdit := Status_GVL.Edit[3],
    bUpload := Status_GVL.Upload[3],
    bDownload := Status_GVL.Download[3],
    bSave := Status_GVL.Save[3],
    bCancel := Status_GVL.Cancel[3],
    iRecipeNumber := Status_GVL.RecipeNumber[3],
    stDataHMI := HMI_GVL.arRecipeHMI[3],
    stPLCRecipe := Status_GVL.arProductList,
    stDataToRobot := Status_GVL.RecipeLine[3],
    stOffsetPattern := Status_GVL.OffsetPattern3,
    HMI_OffsetPattern := HMI_GVL.OffsetPattern3,
    Robot_ProductLength => InputOutput_GVL.xOut_Robot.LengthL3.nUINT,
    Robot_ProductWidth => InputOutput_GVL.xOut_Robot.WidthL3.nUINT,
    Robot_ProductHeight => InputOutput_GVL.xOut_Robot.HeightL3.nUINT,
    Robot_ProductPattern => InputOutput_GVL.xOut_Robot.PatternL3); // FB_Recipe
Status_GVL.StsEdit[3] := NOT Recipe_3.bStsEditMode;

// NETWORK 11
CustomPattern_3(
    ENI := TRUE,
    CycleAtLayer := Status_GVL.CycleAtLayer[3],
    dtRecipe := Status_GVL.RecipeLine[3],
    Offset_X => InputOutput_GVL.xOut_Robot.CustomX3.nUINT,
    Offset_Y => InputOutput_GVL.xOut_Robot.CustomY3.nUINT); // RobotCustomPattern

// NETWORK 12
Layer_3(
    ENI := TRUE,
    CounterCycle := HMI_GVL.arCountPlace[3],
    PatternNumber := Status_GVL.RecipeLine[3].ProductPattern,
    CurrentLayer => Status_GVL.CurrentLayer[3],
    QtyCyclePerLayer => Status_GVL.QtyCyclePerLayer[3],
    CycleAtLayer => Status_GVL.CycleAtLayer[3]); // FB_Layer

// NETWORK 13 (disabled)
// label: Recipe Line 4

// NETWORK 14
Recipe_4(
    ENI := TRUE,
    bEdit := Status_GVL.Edit[4],
    bUpload := Status_GVL.Upload[4],
    bDownload := Status_GVL.Download[4],
    bSave := Status_GVL.Save[4],
    bCancel := Status_GVL.Cancel[4],
    iRecipeNumber := Status_GVL.RecipeNumber[4],
    stDataHMI := HMI_GVL.arRecipeHMI[4],
    stPLCRecipe := Status_GVL.arProductList,
    stDataToRobot := Status_GVL.RecipeLine[4],
    stOffsetPattern := Status_GVL.OffsetPattern4,
    HMI_OffsetPattern := HMI_GVL.OffsetPattern4,
    Robot_ProductLength => InputOutput_GVL.xOut_Robot.LengthL4.nUINT,
    Robot_ProductWidth => InputOutput_GVL.xOut_Robot.WidthL4.nUINT,
    Robot_ProductHeight => InputOutput_GVL.xOut_Robot.HeightL4.nUINT,
    Robot_ProductPattern => InputOutput_GVL.xOut_Robot.PatternL4); // FB_Recipe
Status_GVL.StsEdit[4] := NOT Recipe_4.bStsEditMode;

// NETWORK 15
CustomPattern_4(
    ENI := TRUE,
    CycleAtLayer := Status_GVL.CycleAtLayer[4],
    dtRecipe := Status_GVL.RecipeLine[4],
    Offset_X => InputOutput_GVL.xOut_Robot.CustomX4.nUINT,
    Offset_Y => InputOutput_GVL.xOut_Robot.CustomY4.nUINT); // RobotCustomPattern

// NETWORK 16
Layer_4(
    ENI := TRUE,
    CounterCycle := HMI_GVL.arCountPlace[4],
    PatternNumber := Status_GVL.RecipeLine[4].ProductPattern,
    CurrentLayer => Status_GVL.CurrentLayer[4],
    QtyCyclePerLayer => Status_GVL.QtyCyclePerLayer[4],
    CycleAtLayer => Status_GVL.CycleAtLayer[4]); // FB_Layer

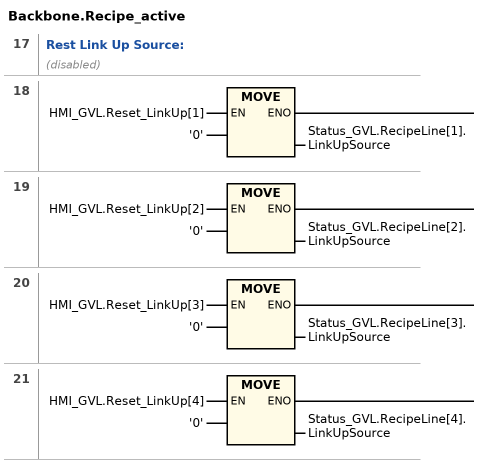
// NETWORK 17 (disabled)
// label: Rest Link Up Source

// NETWORK 18
IF HMI_GVL.Reset_LinkUp[1] THEN Status_GVL.RecipeLine[1].LinkUpSource := '0'; END_IF

// NETWORK 19
IF HMI_GVL.Reset_LinkUp[2] THEN Status_GVL.RecipeLine[2].LinkUpSource := '0'; END_IF

// NETWORK 20
IF HMI_GVL.Reset_LinkUp[3] THEN Status_GVL.RecipeLine[3].LinkUpSource := '0'; END_IF

// NETWORK 21
IF HMI_GVL.Reset_LinkUp[4] THEN Status_GVL.RecipeLine[4].LinkUpSource := '0'; END_IF
END_ACTION

ACTION RTC_Management_active:
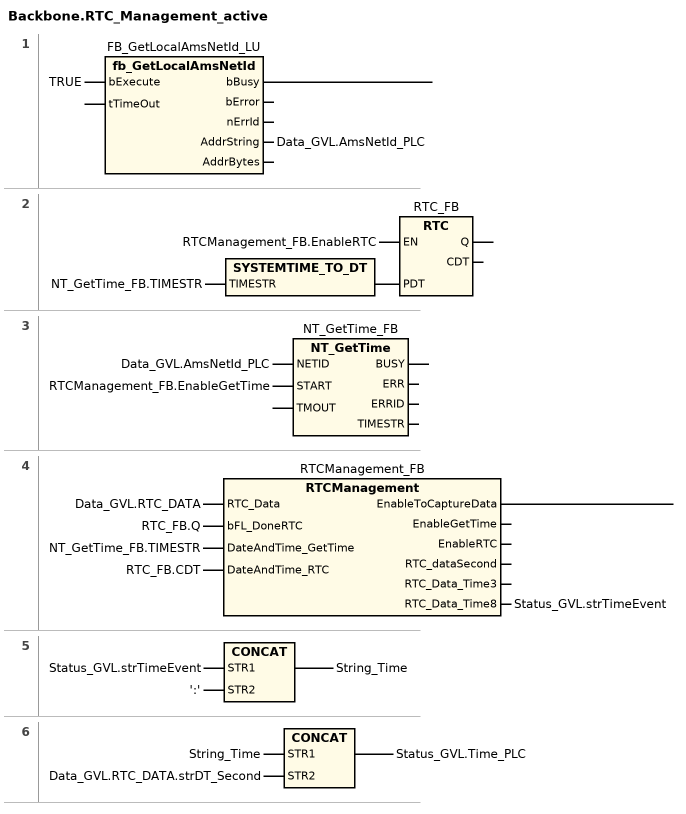
// NETWORK 1
FB_GetLocalAmsNetId_LU(bExecute := TRUE, AddrString => Data_GVL.AmsNetId_PLC); // fb_GetLocalAmsNetId

// NETWORK 2
RTC_FB(EN := RTCManagement_FB.EnableRTC, PDT := SYSTEMTIME_TO_DT(TIMESTR := NT_GetTime_FB.TIMESTR)); // RTC

// NETWORK 3
NT_GetTime_FB(NETID := Data_GVL.AmsNetId_PLC, START := RTCManagement_FB.EnableGetTime); // NT_GetTime

// NETWORK 4
RTCManagement_FB(
    RTC_Data := Data_GVL.RTC_DATA,
    bFL_DoneRTC := RTC_FB.Q,
    DateAndTime_GetTime := NT_GetTime_FB.TIMESTR,
    DateAndTime_RTC := RTC_FB.CDT,
    RTC_Data_Time8 => Status_GVL.strTimeEvent); // RTCManagement

// NETWORK 5
String_Time := CONCAT(STR1 := Status_GVL.strTimeEvent, STR2 := ':');

// NETWORK 6
Status_GVL.Time_PLC := CONCAT(STR1 := String_Time, STR2 := Data_GVL.RTC_DATA.strDT_Second);
END_ACTION

ACTION Test_Outfeed_active:
(**============= Note ================*)
//InputOutput_GVL.TestMode[100] ==> Download Parameter Shuttle Position	
//InputOutput_GVL.TestMode[99]	==> Status Safety
//InputOutput_GVL.TestMode[98]	==> Mute Buzzer
//InputOutput_GVL.TestMode[97]	==> Disable Overflow
//InputOutput_GVL.TestMode[96]	==> Lock Modullar To Run;
//InputOutput_GVL.TestMode[95]	==> Acknowledge Button
//InputOutput_GVL.TestMode[94]	==> Reset Button
//InputOutput_GVL.TestMode[93]	==> Status Running Picking
//InputOutput_GVL.TestMode[92]	==> Bypass Wrapper
//InputOutput_GVL.TestMode[91]	==> Bypass Wrapper Existing


(**============= Test Mode Outfeed ================*)
//=====> Outfeed
InputOutput_GVL.TestMode[1]							:= HMI_GVL.Test_PalletBuffer2_Fwd;
InputOutput_GVL.TestMode[2]							:= HMI_GVL.Test_PalletBuffer1_Fwd;
InputOutput_GVL.TestMode[3]							:= HMI_GVL.Test_PalletOutfeed1_Fwd;
InputOutput_GVL.TestMode[4]							:= HMI_GVL.Test_PalletOutfeed2_Fwd;
InputOutput_GVL.TestMode[5]							:= HMI_GVL.Test_PalletOutfeed3_Fwd;
InputOutput_GVL.TestMode[6]							:= HMI_GVL.Test_PalletOutfeed4_Fwd;
InputOutput_GVL.TestMode[7]							:= HMI_GVL.Test_PalletOutfeed5_Fwd;
InputOutput_GVL.TestMode[8]							:= HMI_GVL.Test_PalletRALifter;
InputOutput_GVL.TestMode[9]							:= HMI_GVL.Test_PalletRATransfer;

IF InputOutput_GVL.Outfeed_stsMachine <> 'Manual' THEN
	HMI_GVL.Test_PalletBuffer2_Fwd					:= FALSE;
	HMI_GVL.Test_PalletBuffer1_Fwd					:= FALSE;
	HMI_GVL.Test_PalletOutfeed1_Fwd					:= FALSE;
	HMI_GVL.Test_PalletOutfeed2_Fwd					:= FALSE;
	HMI_GVL.Test_PalletOutfeed3_Fwd					:= FALSE;
	HMI_GVL.Test_PalletOutfeed4_Fwd					:= FALSE;
	HMI_GVL.Test_PalletOutfeed5_Fwd					:= FALSE;
END_IF

//=====> Shuttle
InputOutput_GVL.TestMode[10]						:= HMI_GVL.Test_ShuttleDrive_Fwd;
InputOutput_GVL.TestMode[11]						:= HMI_GVL.Test_ShuttleDrive_Rev;
InputOutput_GVL.TestMode[12]						:= HMI_GVL.Test_ShuttleLoad_Fwd;
InputOutput_GVL.TestMode[13]						:= HMI_GVL.Test_ShuttleLoad_Rev;
InputOutput_GVL.TestMode[14]						:= HMI_GVL.Test_ShuttleEmpty_Fwd;

IF InputOutput_GVL.Shuttle_stsMachine <> 'Manual' THEN
	HMI_GVL.Test_ShuttleDrive_Fwd					:= FALSE;
	HMI_GVL.Test_ShuttleDrive_Rev					:= FALSE;
	HMI_GVL.Test_ShuttleLoad_Fwd					:= FALSE;
	HMI_GVL.Test_ShuttleLoad_Rev					:= FALSE;
	HMI_GVL.Test_ShuttleEmpty_Fwd					:= FALSE;
END_IF

//=====> Infeed
InputOutput_GVL.TestMode[15]						:= HMI_GVL.Test_BoxInfeed_Fwd;
InputOutput_GVL.TestMode[16]						:= HMI_GVL.Test_BoxStopGo_Fwd;
InputOutput_GVL.TestMode[17]						:= HMI_GVL.Test_BoxBuffer1_Fwd;
InputOutput_GVL.TestMode[18]						:= HMI_GVL.Test_BoxBuffer2_Fwd;
InputOutput_GVL.TestMode[19]						:= HMI_GVL.Test_BoxModullar1_Fwd;
InputOutput_GVL.TestMode[20]						:= HMI_GVL.Test_BoxModullar2_Fwd;
InputOutput_GVL.TestMode[21]						:= HMI_GVL.Test_BoxModullar3_Fwd;
InputOutput_GVL.TestMode[22]						:= HMI_GVL.Test_BoxModullar4_Fwd;
InputOutput_GVL.TestMode[23]						:= HMI_GVL.Test_Stopper1;
InputOutput_GVL.TestMode[24]						:= HMI_GVL.Test_Stopper2;
InputOutput_GVL.TestMode[25]						:= HMI_GVL.Test_Pusher_StopGo_Adv;
InputOutput_GVL.TestMode[26]						:= HMI_GVL.Test_Pusher_StopGo_Rtc;
InputOutput_GVL.TestMode[27]						:= HMI_GVL.Test_Pusher_Buffer1_Adv;
InputOutput_GVL.TestMode[28]						:= HMI_GVL.Test_Pusher_Buffer1_Rtc;
InputOutput_GVL.TestMode[29]						:= HMI_GVL.Test_Pusher_Buffer2_Adv;
InputOutput_GVL.TestMode[30]						:= HMI_GVL.Test_Pusher_Buffer2_Rtc;
InputOutput_GVL.TestMode[31]						:= HMI_GVL.Test_StopperModullar_Adv;
InputOutput_GVL.TestMode[32]						:= HMI_GVL.Test_StopperModullar_Rtc;

IF InputOutput_GVL.Infeed_stsMachine <> 'Manual' THEN
	HMI_GVL.Test_BoxInfeed_Fwd						:= FALSE;
	HMI_GVL.Test_BoxStopGo_Fwd						:= FALSE;
	HMI_GVL.Test_BoxBuffer1_Fwd						:= FALSE;
	HMI_GVL.Test_BoxBuffer2_Fwd						:= FALSE;
	HMI_GVL.Test_BoxModullar1_Fwd					:= FALSE;
	HMI_GVL.Test_BoxModullar2_Fwd					:= FALSE;
	HMI_GVL.Test_BoxModullar3_Fwd					:= FALSE;
	HMI_GVL.Test_BoxModullar4_Fwd					:= FALSE;
	HMI_GVL.Test_Stopper1							:= FALSE;
	HMI_GVL.Test_Stopper2							:= FALSE;
	HMI_GVL.Test_Pusher_StopGo_Adv					:= FALSE;
	HMI_GVL.Test_Pusher_StopGo_Rtc					:= FALSE;
	HMI_GVL.Test_Pusher_Buffer1_Adv					:= FALSE;
	HMI_GVL.Test_Pusher_Buffer1_Rtc					:= FALSE;
	HMI_GVL.Test_Pusher_Buffer2_Adv					:= FALSE;
	HMI_GVL.Test_Pusher_Buffer2_Rtc					:= FALSE;
END_IF
END_ACTION

END_PROGRAM

// ---- POUs/Function_Block/General/RTCManagement.TcPOU
FUNCTION_BLOCK RTCManagement
VAR_IN_OUT
	RTC_Data 			: stRTC_Data;
END_VAR
VAR_INPUT
	bFL_DoneRTC			: BOOL;
	DateAndTime_GetTime	: TIMESTRUCT;
	DateAndTime_RTC		: DT;
END_VAR
VAR_OUTPUT
	EnableToCaptureData	: BOOL;	
	EnableGetTime		: BOOL;
	EnableRTC			: BOOL;
	RTC_dataSecond 		: INT ;
	RTC_Data_Time8 		: STRING;
END_VAR
VAR

	RealTimeClock		: RTC;
	DateAndTime			: TIMESTRUCT;
	SeqIndex			: INT;
	
	wYear				: INT;
	Input_RTC			: DATE_AND_TIME;
	
	RTC_Data_Time1 		: STRING;
	RTC_Data_Time2 		: STRING;
	RTC_Data_Time3 		: STRING;
	RTC_Data_Time4 		: STRING;
	RTC_Data_Time5 		: STRING;
	RTC_Data_Time6 		: STRING;
	RTC_Data_Time7 		: STRING;
	
END_VAR

(*======================FB RTC MANAGEMENT V0.1================*)
// Changelog[ 22/09/2022] M.Dimas Andiwjaya 



CASE SeqIndex OF
	0:
		EnableGetTime:=TRUE;
		IF NOT (DateAndTime_GetTime.wYear=0) THEN
			SeqIndex:=10;
		END_IF
	10:
		EnableGetTime:=FALSE;
		Input_RTC:=SYSTEMTIME_TO_DT(DateAndTime_GetTime);
		EnableRTC:=TRUE;
		IF bFL_DoneRTC THEN
			SeqIndex:=20;
		END_IF
	20:
		DateAndTime:=DT_TO_SYSTEMTIME(DateAndTime_RTC);
		RTC_Data.iDT_Year	:=WORD_TO_INT(DateAndTime.wYear);
		RTC_Data.iDT_Month	:=WORD_TO_INT(DateAndTime.wMonth);
		RTC_Data.iDT_Date	:=WORD_TO_INT(DateAndTime.wDay);
		RTC_Data.iDT_Hour	:=WORD_TO_INT(DateAndTime.wHour);
		RTC_Data.iDT_Minute	:=WORD_TO_INT(DateAndTime.wMinute);
		RTC_Data.iDT_Second	:=WORD_TO_INT(DateAndTime.wSecond);	
		RTC_dataSecond := RTC_Data.iDT_Second ;
		RTC_Data.iDT_MilliSecond	:=WORD_TO_INT(DateAndTime.wMilliseconds);
	
		RTC_Data.strDT_MilliSecond := INT_TO_STRING(RTC_Data.iDT_MilliSecond);
		IF RTC_Data.iDT_Second <= 9 THEN
			RTC_Data.strDT_Second:=CONCAT('0',INT_TO_STRING(RTC_Data.iDT_Second));
		ELSE
			RTC_Data.strDT_Second:=INT_TO_STRING(RTC_Data.iDT_Second);
		END_IF
		
		IF RTC_Data.iDT_Minute <= 9 THEN
			RTC_Data.strDT_Minute:=CONCAT('0',INT_TO_STRING(RTC_Data.iDT_Minute));
		ELSE
			RTC_Data.strDT_Minute:=INT_TO_STRING(RTC_Data.iDT_Minute);
		END_IF
		
		IF RTC_Data.iDT_Hour <= 9 THEN
			RTC_Data.strDT_Hour:=CONCAT('0',INT_TO_STRING(RTC_Data.iDT_Hour));
		ELSE
			RTC_Data.strDT_Hour:=INT_TO_STRING(RTC_Data.iDT_Hour);
		END_IF
		
		RTC_Data.strDT_Year := INT_TO_STRING (RTC_Data.iDT_Year);
		
		IF RTC_Data.iDT_Month <= 9 THEN
			RTC_Data.strDT_Month:=CONCAT('0',INT_TO_STRING(RTC_Data.iDT_Month));
		ELSE
			RTC_Data.strDT_Month:=INT_TO_STRING(RTC_Data.iDT_Month);
		END_IF
		IF RTC_DATA.iDT_Date <=9 THEN 
			RTC_Data.strDT_Date:=CONCAT('0',INT_TO_STRING(RTC_Data.iDT_Date));
		ELSE
			RTC_Data.strDT_Date:=INT_TO_STRING(RTC_Data.iDT_Date);
		END_IF
		RTC_Data_Time1 := Concat(':',RTC_Data.strDT_Minute);
		RTC_Data_Time2 := Concat(RTC_Data.strDT_Hour,RTC_Data_Time1);
		RTC_Data_Time3 := concat(' ',RTC_Data_Time2);
		RTC_Data_Time4 := Concat(RTC_Data.strDT_Year,RTC_Data_Time3);
		RTC_Data_Time5 := Concat ('/',RTC_Data_Time4);
		RTC_Data_Time6 := Concat(RTC_Data.strDT_Month,RTC_Data_Time5);
		RTC_Data_Time7 := Concat('/',RTC_Data_Time6);
		RTC_Data_Time8 := concat (RTC_Data.strDT_Date,RTC_Data_Time7);
END_CASE

END_FUNCTION_BLOCK

// ---- POUs/Function_Block/Robot/FB_Recipe.TcPOU
FUNCTION_BLOCK FB_Recipe
VAR_INPUT
	ENI						: BOOL;
	bEdit					: BOOL;
	bUpload					: BOOL;
	bDownload				: BOOL;
	bSave					: BOOL;
	bCancel					: BOOL;
END_VAR
VAR_OUTPUT
	ENO						: BOOL;
	bStsEditMode			: BOOL;
	iSelectedRecipeNumber	: USINT;
	Robot_ProductLength		: UINT;
	Robot_ProductWidth		: UINT;
	Robot_ProductHeight		: UINT;
	Robot_ProductPattern	: USINT;
END_VAR

VAR
	Temp_Data1				: stProductInfo;
	DataTimer				: TON;
	TempRecipeNumber		: USINT;
END_VAR

VAR_IN_OUT
	iRecipeNumber			: USINT;
	stDataHMI				: stProductInfo;
	stPLCRecipe				: ARRAY[1..40] OF stProductInfo;
	stDataToRobot			: stProductInfo;
	stOffsetPattern			: ARRAY[1..40] OF stCustomPattern;
	HMI_OffsetPattern		: stCustomPattern;
END_VAR

//=======FB_Recipe v1.0=======
//Used UDTs: sProductInfo - v3.0
//

//Changelog
//v1.0 Add bStsEditMode & bStsCopyMode
//v2.0 Without Barcode
//v3.0 Add In/Out Offset Pattern

//==================================

IF ENI THEN
	ENO:=TRUE;
END_IF;


IF iRecipeNumber < 1  THEN
	iRecipeNumber:=40;
END_IF;
IF iRecipeNumber > 40 THEN
	iRecipeNumber:=1;
END_IF;



IF bStsEditMode THEN
	Temp_Data1				:= stDataHMI;
	//Temp_Data1.ProductName	:= sProductName;
	IF bUpload THEN
		stDataHMI			:= stDataToRobot;
	ELSIF bSave THEN
		stPLCRecipe[iRecipeNumber]		:= stDataHMI;
		stOffsetPattern[iRecipeNumber]	:= stDataHMI.OffsetPattern;
		bStsEditMode					:= FALSE;
	END_IF;
ELSE
	stDataHMI				:= stPLCRecipe[iRecipeNumber];
	stDataHMI.OffsetPattern := stOffsetPattern[iRecipeNumber];
	//sProductName			:= stPLCRecipe[iRecipeNumber].ProductName;
	
	IF bDownload THEN
		//stDataToRobot.ProductName:='                                 ';
		//IF stDataToRobot.ProductName='                                 ' THEN
			//stDataToRobot				:= stPLCRecipe[iRecipeNumber];
			stDataToRobot.ProductName	:= stPLCRecipe[iRecipeNumber].ProductName;
			stDataToRobot.ProductLength	:= stPLCRecipe[iRecipeNumber].ProductLength;
			stDataToRobot.ProductWidth	:= stPLCRecipe[iRecipeNumber].ProductWidth;
			stDataToRobot.ProductHeight	:= stPLCRecipe[iRecipeNumber].ProductHeight;
			stDataToRobot.ProductPattern:= stPLCRecipe[iRecipeNumber].ProductPattern;
			stDataToRobot.Stacking		:= stPLCRecipe[iRecipeNumber].Stacking;
			stDataToRobot.LinkUpSource	:= stPLCRecipe[iRecipeNumber].LinkUpSource;
			stDataToRobot.OffsetPattern := stOffsetPattern[iRecipeNumber];
			iSelectedRecipeNumber		:= iRecipeNumber;
		//END_IF;
	END_IF;
END_IF;

IF iRecipeNumber<> TempRecipeNumber THEN
	//sProductName:='                                 ';
	TempRecipeNumber := iRecipeNumber;
END_IF;

IF bEdit THEN
	bStsEditMode := TRUE;
END_IF;

IF bCancel THEN
	bStsEditMode := FALSE;
END_IF;


Robot_ProductLength		:= stDataToRobot.ProductLength;
Robot_ProductWidth		:= stDataToRobot.ProductWidth;
Robot_ProductHeight		:= stDataToRobot.ProductHeight;
Robot_ProductPattern	:= stDataToRobot.ProductPattern;

END_FUNCTION_BLOCK

// ---- POUs/Function_Block/Robot/RobotCustomPattern.TcPOU
FUNCTION_BLOCK RobotCustomPattern
VAR_INPUT
	ENI				: BOOL;
	CycleAtLayer	: UINT;
	dtRecipe		: stProductinfo;
END_VAR
VAR_OUTPUT
	ENO				: BOOL;
	Offset_X		: UINT;
	Offset_Y		: UINT;
	Offset_Z		: UINT;
END_VAR

VAR
	
END_VAR

IF ENI THEN
	ENO:=TRUE;
	
	
	IF CycleAtLayer <> 0 THEN
		Offset_X := INT_TO_UINT(dtRecipe.OffsetPattern.Offset_X[CycleAtLayer]);
		Offset_Y := INT_TO_UINT(dtRecipe.OffsetPattern.Offset_Y[CycleAtLayer]);
		Offset_Z := INT_TO_UINT(dtRecipe.OffsetPattern.Offset_Z[CycleAtLayer]);
	END_IF
	
	
	
END_IF;

END_FUNCTION_BLOCK

// ---- POUs/Function_Block/Robot/FB_Layer.TcPOU
FUNCTION_BLOCK FB_Layer
VAR_INPUT
	ENI				: BOOL;
	CounterCycle	: UINT;
	PatternNumber	: UINT;
END_VAR
VAR_OUTPUT
	ENO				: BOOL;
	CurrentLayer	: UINT;
	QtyCyclePerLayer: UINT;
	CycleAtLayer	: UINT;
END_VAR

VAR
	
END_VAR

IF ENI THEN
	ENO 	:= TRUE;
	
	//Quantity Cycle Per Layer
	CASE PatternNumber OF
		1:	QtyCyclePerLayer	:= 9;	//Japan Box
		2:	QtyCyclePerLayer	:= 10;	//Standard 
		3:	QtyCyclePerLayer	:= 12;	//Small LU18
		4:	QtyCyclePerLayer	:= 7;	//Small LU26
		0:	QtyCyclePerLayer	:= 1;
	END_CASE 
	
	//Current Layer
	CurrentLayer	:= ((CounterCycle - 1)/QtyCyclePerLayer)+1;

	//Cycle at Current Layer
	CycleAtLayer := CounterCycle MOD (2*QtyCyclePerLayer);
	IF CycleAtLayer = 0 AND CounterCycle <> 0 THEN
		CycleAtLayer := 2*QtyCyclePerLayer;
	END_IF;
	
END_IF;

END_FUNCTION_BLOCK

// ---- POUs/Function_Block/General/FGHS_DataCollect_Palletizing.TcPOU
FUNCTION_BLOCK FGHS_DataCollect_Palletizing

VAR_INPUT
	ENI					: BOOL;
	bResetBuffer		: BOOL;
	bReset				: BOOL;
	bHandshake			: BOOL;
	bDonePick			: BOOL;
	bDonePlace			: BOOL;	
	iCycleBox			: UINT;
	iLine				: STRING;
	Barcode				: STRING;
	PalletID			: STRING;	
	Timestamp			: DT;
	ProductData			: stProductInfo;
END_VAR


VAR_OUTPUT
	ENO					: BOOL;
	Error				: BOOL;
	ErrorMsg			: STRING;
	DoneScan			: BOOL;
END_VAR

VAR_IN_OUT
	arBuffer			: stPalletTrackingData;
END_VAR

VAR PERSISTENT
	EmptyArray			: stPalletTrackingData;
	TempBarcode			: STRING;
	DataTimer			: TON;
	R_DonePlace			: R_TRIG;
	R_DonePick			: R_TRIG;
	T_DonePick			: TOF;
	SeqIndex			: INT;
	SeqIndex2			: INT;
	Index				: UINT;
	LastCycle			: UINT;
	BarcodeEAN			: STRING;
	CodeVariant			: STRING;
	BarcodeLinkUp		: STRING;
	BarcodeResult		: STRING;
END_VAR

IF ENI THEN
	ENO	:= TRUE;
END_IF
IF bReset THEN
	Error 		:= FALSE;
	ErrorMsg	:= '';
END_IF


//Get Data Barcode at Picking to Temp Variable
CASE SeqIndex OF 
	0:
		DoneScan	:= FALSE;
		IF bDonePick THEN
			SeqIndex	:= 1;
		END_IF
		
	1:
		TempBarcode	:= Barcode;
		DoneScan	:= TRUE;
		//IF arBuffer.BarcodeProduct[iCycleBox] = TempBarcode THEN
		//	Warning	:= TRUE;
		//END_IF
		
		IF NOT bDonePick THEN
			SeqIndex	:= 0;
		END_IF
		
		
END_CASE

//Get Data Barcode and Timestamp when Product Placed at Pallet
R_DonePlace(CLK:= bDonePlace);
IF R_DonePlace.Q THEN
	arBuffer.BarcodeProduct[iCycleBox]		:= TempBarcode;
	arBuffer.BarcodeProductTime[iCycleBox]	:= Timestamp;
	
	
	
END_IF


//Move Pallet ID 
IF iCycleBox > 1 AND PalletID <> '' THEN
	arBuffer.PalletID			:= PalletID;
	arBuffer.PalletCreationDate	:= Timestamp;
	arBuffer.EANVariant			:= ProductData.EANVariant;
	arBuffer.CodeVariant		:= ProductData.CodeVariant;
	arBuffer.CounterProduct		:= iCycleBox-1;
ELSIF (PalletID = '' AND bHandshake) OR bResetBuffer THEN //
	arBuffer					:= EmptyArray;
END_IF


IF iCycleBox > 1 THEN
	//Detect Dupilcate Barcode
	IF arBuffer.BarcodeProduct[iCycleBox] = arBuffer.BarcodeProduct[iCycleBox-1] THEN // OR (R_DonePick.Q AND TempBarcode = arBuffer.BarcodeProduct[iCycleBox-1])) AND arBuffer.BarcodeProduct[iCycleBox-1] <> ''
		Error		:= TRUE;
		ErrorMsg	:= CONCAT('Duplicate Barcode at Placing ',iLine);
	END_IF	
	
	(* Split Barcode *)
	BarcodeResult	:= arBuffer.BarcodeProduct[iCycleBox-1];
	BarcodeEAN		:= DELETE(DELETE(BarcodeResult,3,0),24,15);
	CodeVariant		:= DELETE(DELETE(BarcodeResult,19,0),20,3);
	BarcodeLinkUp	:= DELETE(DELETE(BarcodeResult,33,0),6,3);
	
	//Detect Misplaced Barcode
	IF ProductData.LinkUpSource <> BarcodeLinkUp AND BarcodeResult <> '' AND (ProductData.LinkUpSource <> '0' OR ProductData.LinkUpSource <> '') THEN
		Error		:= TRUE;
		ErrorMsg	:= CONCAT('Mixing Barcode at Placing ',iLine);
	END_IF 
	
END_IF



//Release Barcode 
IF LastCycle <> iCycleBox AND iCycleBox > 1 AND PalletID <> '' AND NOT ENI THEN
	FOR Index := iCycleBox+1 TO 60 BY 1 DO	
		arBuffer.BarcodeProduct[Index]		:= EmptyArray.BarcodeProduct[Index];
		arBuffer.BarcodeProductTime[Index]	:= EmptyArray.BarcodeProductTime[Index];
	END_FOR
	LastCycle	:= iCycleBox;
END_IF

END_FUNCTION_BLOCK

// ---- POUs/Function_Block/General/Alarm_Event_History.TcPOU
FUNCTION_BLOCK Alarm_Event_History

VAR_INPUT
	bError			: BOOL;
	bErrorID		: UINT;
	strErrorMsg		: STRING;
	TimeStop		: STRING;	
	bResetBuffer	: BOOL;
END_VAR
VAR_OUTPUT
	bEnable_Out		: BOOL;
END_VAR
VAR
	EmptyArray 		: INT ;
	temp 			: INT ;
	leght 			: INT := 100;
	rTrig_Error 	: R_TRIG;
	j				: INT;
END_VAR
VAR_IN_OUT
	dtErrorHistory	: ARRAY [0..100] OF stErrorData;
END_VAR

(*
	=============FB Error History V0.1===========
*)
rTrig_Error(clk:= bError);
bEnable_Out := NOT bError;

     IF rTrig_Error.Q THEN 
    // Memulai perekaman data kesalahan baru saat terjadi kesalahan baru
       dtErrorHistory[0].Status      := 1;            // Set status entri kesalahan sebagai aktif
       dtErrorHistory[0].ErrorID     := bErrorID;    // Simpan ID kesalahan
       dtErrorHistory[0].ErrorMsg    := strErrorMsg;    // Simpan pesan kesalahan
       dtErrorHistory[0].TimeStop    := TimeStop;    // Simpan waktu terjadinya kesalahan

    // Geser data kesalahan lama ke posisi yang lebih tinggi dalam array
       temp := leght;
       FOR EmptyArray := 1 TO leght BY 1 DO 
          dtErrorHistory[temp].Status        := dtErrorHistory[temp-1].Status ;
          dtErrorHistory[temp].ErrorID       := dtErrorHistory[temp-1].ErrorID ;
          dtErrorHistory[temp].ErrorMsg      := dtErrorHistory[temp-1].ErrorMsg ;
          dtErrorHistory[temp].TimeStop      := dtErrorHistory[temp-1].TimeStop ;
          temp := temp-1;
       END_FOR

    // Menetapkan nilai kosong untuk entri kesalahan terbaru
       dtErrorHistory[0].Status      := 0;
       dtErrorHistory[0].ErrorID     := 0;
       dtErrorHistory[0].ErrorMsg    := '';
       dtErrorHistory[0].TimeStop    := '';
     END_IF 

	
     IF dtErrorHistory[100].Status = 1 THEN
    // Jika entri kesalahan terakhir menunjukkan status aktif
    // Artinya buffer kesalahan sudah penuh, maka lakukan pembersihan
        FOR j := 1  TO leght BY 1 DO 
        // Reset nilai-nilai dalam setiap entri array untuk membersihkan riwayat kesalahan
           dtErrorHistory[j].Status      := 0;
           dtErrorHistory[j].ErrorID     := 0;
           dtErrorHistory[j].ErrorMsg    := '';
           dtErrorHistory[j].TimeStop    := '';
        END_FOR
     END_IF

END_FUNCTION_BLOCK

// ---- POUs/Function_Block/General/Alarm_Event_Active.TcPOU
FUNCTION_BLOCK Alarm_Event_Active

VAR_INPUT
	bError			: BOOL;
	bErrorID		: UINT;
	strErrorMsg		: STRING;
	TimeStop		: STRING;	
	bResetBuffer	: BOOL;
END_VAR
VAR_OUTPUT
	bEnable_Out		: BOOL;
END_VAR
VAR
	EmptyArray 		: INT ;
	temp 			: INT ;
	leght 			: INT := 100;
	rTrig_Error 	: R_TRIG;
	fTrig_Error 	: F_TRIG;
	i				: INT;
	Seq				: INT;
	IndexReset		: INT;
	Cycle			: INT;
	EmptyBuffer		: ARRAY [0..100] OF stErrorData;
	bReset			: BOOL;
END_VAR
VAR_IN_OUT
	dtError			: ARRAY [0..100] OF stErrorData;
END_VAR

(*
	=============FB Error History V0.1===========
*)
(*IF bReset THEN
	dtError		:= EmptyBuffer;
END_IF

rTrig_Error(clk:= bError);
bEnable_Out := NOT bError;
	IF  rTrig_Error.Q AND dtError[1].ErrorID <> bErrorID THEN 
		
		dtError[0].Status	:= 1;
		dtError[0].ErrorID	:= bErrorID;
		dtError[0].ErrorMsg	:= strErrorMsg;
		dtError[0].TimeStop	:= TimeStop;
		temp := leght;
		FOR EmptyArray := 1 TO leght BY 1 DO 
			dtError[temp].Status	:= dtError[temp-1].Status ;
			dtError[temp].ErrorID	:= dtError[temp-1].ErrorID ;
			dtError[temp].ErrorMsg	:= dtError[temp-1].ErrorMsg ;
			dtError[temp].TimeStop	:= dtError[temp-1].TimeStop ;
			temp := temp-1;
		END_FOR
		dtError[0].Status	:= 0;
		dtError[0].ErrorID	:= 0;
		dtError[0].ErrorMsg	:= '';
		dtError[0].TimeStop	:= '';
 	END_IF 
	
fTrig_Error(clk:= bError);
CASE Seq OF
	0:
		IF (NOT bError AND bResetBuffer) THEN //OR fTrig_Error.Q 
			Seq	:= 1;
		END_IF
		
	1:
		i:=0;
		FOR i := 1 TO leght BY 1 DO
			IF dtError[i].ErrorID = bErrorID AND dtError[i].ErrorID <> 0 THEN
				IndexReset	:= i;
				Seq			:= 2;
				EXIT;
			END_IF
		END_FOR 
		IF i > leght THEN
			Seq	:= 0;
		END_IF
		
	
	2:
		i:=0;
		FOR i := IndexReset TO leght BY 1 DO
				dtError[i].Status		:= dtError[i+1].Status ;
				dtError[i].ErrorID		:= dtError[i+1].ErrorID ;
				dtError[i].ErrorMsg		:= dtError[i+1].ErrorMsg ;
				dtError[i].TimeStop		:= dtError[i+1].TimeStop ;
		END_FOR 
		
		IF i > leght THEN
			Seq	:= 1;
		END_IF
		
	
		
	3:
		IF NOT fTrig_Error.Q AND NOT bResetBuffer THEN 
			Seq	:= 0;
		END_IF
		
END_CASE
*)

(*
    =========================================================
    FB Error History V0.1
    =========================================================
    Deskripsi:
    Program ini bertanggung jawab untuk merekam, menyimpan, 
    dan mengelola riwayat peristiwa kesalahan dalam sistem PLC.
*)

IF bReset THEN
    // Jika sinyal reset diaktifkan, reset buffer kesalahan
    dtError    := EmptyBuffer;
END_IF

// Pemicu yang diatur berdasarkan sinyal bError
rTrig_Error(clk:= bError);
// Output bEnable_Out merupakan negasi dari sinyal bError
bEnable_Out := NOT bError;

IF  rTrig_Error.Q AND dtError[1].ErrorID <> bErrorID THEN 
    // Jika terjadi peristiwa kesalahan baru
    // Simpan informasi kesalahan dalam entri pertama array
    dtError[0].Status      := 1;            // Status aktif
    dtError[0].ErrorID     := bErrorID;    // ID kesalahan
    dtError[0].ErrorMsg    := strErrorMsg;    // Pesan kesalahan
    dtError[0].TimeStop    := TimeStop;    // Waktu terjadinya kesalahan

    // Geser data kesalahan lama ke posisi yang lebih tinggi dalam array
    temp := leght;
    FOR EmptyArray := 1 TO leght BY 1 DO 
        dtError[temp].Status        := dtError[temp-1].Status ;
        dtError[temp].ErrorID       := dtError[temp-1].ErrorID ;
        dtError[temp].ErrorMsg      := dtError[temp-1].ErrorMsg ;
        dtError[temp].TimeStop      := dtError[temp-1].TimeStop ;
        temp := temp-1;
    END_FOR

    // Set nilai kosong untuk entri kesalahan terbaru
    dtError[0].Status      := 0;
    dtError[0].ErrorID     := 0;
    dtError[0].ErrorMsg    := '';
    dtError[0].TimeStop    := '';
END_IF 

// Pemicu lain yang diatur berdasarkan sinyal bError
fTrig_Error(clk:= bError);

// Pemrosesan berdasarkan langkah-langkah dalam urutan tertentu
CASE Seq OF
    0:
        // Langkah 0: Menunggu hingga tidak ada kesalahan dan sinyal reset buffer diaktifkan
        IF (NOT bError AND bResetBuffer) THEN 
            Seq    := 1;    // Pindah ke langkah 1
        END_IF
        
    1:
        // Langkah 1: Mencari entri kesalahan yang sesuai dengan ID kesalahan yang baru
        // Jika ditemukan, set langkah selanjutnya
        i:=0;
        FOR i := 1 TO leght BY 1 DO
            IF dtError[i].ErrorID = bErrorID AND dtError[i].ErrorID <> 0 THEN
                IndexReset     := i;    // Simpan indeks untuk langkah selanjutnya
                Seq            := 2;    // Pindah ke langkah 2
                EXIT;
            END_IF
        END_FOR 
        // Jika tidak ditemukan, kembali ke langkah 0
        IF i > leght THEN
            Seq    := 0;
        END_IF
        
    2:
        // Langkah 2: Menghapus entri kesalahan yang sudah ditangani
        i:=0;
        FOR i := IndexReset TO leght BY 1 DO
                // Geser entri kesalahan ke atas untuk menghapus entri yang sudah ditangani
                dtError[i].Status         := dtError[i+1].Status ;
                dtError[i].ErrorID        := dtError[i+1].ErrorID ;
                dtError[i].ErrorMsg       := dtError[i+1].ErrorMsg ;
                dtError[i].TimeStop       := dtError[i+1].TimeStop ;
        END_FOR 
        
        // Jika semua entri kesalahan sudah diproses, kembali ke langkah 1
        IF i > leght THEN
            Seq    := 1;
        END_IF
        
    3:
        // Langkah 3: Menunggu hingga tidak ada kesalahan baru dan reset buffer tidak aktif
        IF NOT fTrig_Error.Q AND NOT bResetBuffer THEN 
            Seq    := 0;    // Kembali ke langkah 0
        END_IF
        
END_CASE

END_FUNCTION_BLOCK

// ---- POUs/Function_Block/General/OEETime.TcPOU
FUNCTION_BLOCK OEETime
VAR_INPUT
	ENI					: BOOL;
	CurrentTime			: DT;
	dt_State			: stMachineState;
	stsMachine			: STRING(31);
END_VAR
VAR_OUTPUT 
	UpTime				: TIME;
END_VAR
VAR_IN_OUT PERSISTENT
	dt_OEE				: sOEETime;
END_VAR
VAR PERSISTENT
	StartedDate			: DATE;
	StartedShift		: UINT;
	dt_TimeCal			: ShiftTime;
	Sts_DailyShiftEnd	: BOOL;
	SaveData			: BOOL;
	bGetData			: BOOL;
	i					: INT;
	j					: INT;
	k					: INT;
	l					: INT;
	m					: INT;
	SeqCal				: INT;
	TimeCal				: TON;
	bTrig				: R_TRIG;
	ShiftDuration		: ARRAY [0..2] OF REAL;
	tUpTime				: TIME;
	Duration			: REAL;
	Time1				: TOD;
	Time2				: TOD;
END_VAR

//Get Time & Parsing
dt_OEE.DateCurrent := DT_TO_DATE(CurrentTime);
dt_OEE.TimeCurrent := DT_TO_TOD(CurrentTime);

dt_OEE.TimeShift[1].StartShift	:= TOD#06:00:00;
dt_OEE.TimeShift[2].StartShift	:= TOD#14:00:00;
dt_OEE.TimeShift[3].StartShift	:= TOD#22:00:00;

dt_OEE.TimeShift[1].EndShift	:= TOD#14:00:00;
dt_OEE.TimeShift[2].EndShift	:= TOD#22:00:00;
dt_OEE.TimeShift[3].EndShift	:= TOD#06:00:00;

//Accumulating Time
CASE SeqCal OF
	0:
			TimeCal(IN:=TRUE, PT:=T#990MS);
			IF TimeCal.Q THEN
				tUpTime	:= tUpTime + T#1S;
				IF  dt_State.Running OR stsMachine = 'Running' THEN
					dt_TimeCal.Running	:= dt_TimeCal.Running + T#1S;
			      	SeqCal							:= 1;
			    ELSIF  dt_State.Error OR dt_State.Aborted OR stsMachine = 'Error' OR stsMachine = 'Aborted' THEN
			        dt_TimeCal.Error	:= dt_TimeCal.Error + T#1S;
			      	SeqCal							:= 1;
			    ELSE //IF NOT  dt_State.Running OR NOT  dt_State.Error OR  dt_State.CheckSafety OR  dt_State.Aborted THEN
			        dt_TimeCal.Stopped	:= dt_TimeCal.Stopped + T#1S;
			      	SeqCal							:= 1;
			    END_IF;
			END_IF;
	1:
			TimeCal(IN:=FALSE);
			SeqCal		:= 0;
	
END_CASE;

Uptime		:= tUpTime;


// Reset Variable Ketika Pergantian Shift
 bTrig(CLK :=  bGetData);
IF  bTrig.Q OR dt_OEE.Reset THEN
     dt_TimeCal.Running		:= T#0s;
	 dt_TimeCal.Error		:= T#0S;
	 dt_TimeCal.Stopped		:= T#0s;
END_IF;



IF (( dt_OEE.TimeCurrent >  dt_OEE.TimeShift[1].EndShift) AND ( dt_OEE.TimeCurrent < dt_OEE.TimeShift[1].EndShift + T#3S)) 
    OR (( dt_OEE.TimeCurrent >  dt_OEE.TimeShift[2].EndShift) AND ( dt_OEE.TimeCurrent < dt_OEE.TimeShift[2].EndShift + T#3S)) 
    OR (( dt_OEE.TimeCurrent >  dt_OEE.TimeShift[3].EndShift) AND ( dt_OEE.TimeCurrent < dt_OEE.TimeShift[3].EndShift + T#3S))  THEN
    IF NOT  bGetData THEN
         bGetData := TRUE;
         StartedDate	:=  dt_OEE.DateCurrent;
         StartedShift	:=  dt_OEE.CurrentShift;
    END_IF;
ELSE
     bGetData := FALSE;
END_IF;

(**Shift Checking**)
IF NOT  SaveData THEN
    IF ( dt_OEE.TimeCurrent >  dt_OEE.TimeShift[1].StartShift) AND ( dt_OEE.TimeCurrent <  dt_OEE.TimeShift[1].EndShift) THEN
         dt_OEE.CurrentShift := 1;
    ELSIF ( dt_OEE.TimeCurrent >  dt_OEE.TimeShift[2].StartShift) AND ( dt_OEE.TimeCurrent <  dt_OEE.TimeShift[2].EndShift) THEN
         dt_OEE.CurrentShift := 2;
    ELSIF ( dt_OEE.TimeCurrent >  dt_OEE.TimeShift[3].StartShift) OR ( dt_OEE.TimeCurrent <  dt_OEE.TimeShift[3].EndShift) THEN
         dt_OEE.CurrentShift := 3;
    END_IF;
END_IF;

(** Function to Clear Data Record **)
(*IF  dt_OEE.Reset THEN
     StartedDate :=  dt_OEE.DateCurrent;
    FOR  l := 1 TO 6 BY 1 DO
        FOR  m := 0 TO 2 BY 1 DO
             dt_OEE.RecordDate[ l] :=  StartedDate;
             dt_OEE.RecordTime[ l,  m].Running   	:= T#0s;
			 dt_OEE.RecordTime[ l,  m].Stopped   	:= T#0s;
			 dt_OEE.RecordTime[ l,  m].Error   		:= T#0s;
             
        END_FOR;
    END_FOR;
        
END_IF;*)

(** Function to copy daily information to history AND Reset Timer**)
IF (( dt_OEE.TimeCurrent >  dt_OEE.TimeShift[3].EndShift) AND ( dt_OEE.TimeCurrent < ( dt_OEE.TimeShift[3].EndShift+T#3S))) AND NOT Sts_DailyShiftEnd THEN
     SaveData := TRUE;
    FOR  i := 5 TO 0 BY -1 DO
        FOR  j := 0 TO 2 BY 1 DO
             dt_OEE.RecordDate[ i + 1]              		:=  dt_OEE.RecordDate[ i];
             dt_OEE.RecordTime[ i + 1,  j].Running 			:=  dt_OEE.RecordTime[ i,  j].Running;
             dt_OEE.RecordTime[ i + 1,  j].Stopped  		:=  dt_OEE.RecordTime[ i,  j].Stopped;
             dt_OEE.RecordTime[ i + 1,  j].Error    		:=  dt_OEE.RecordTime[ i,  j].Error;
        END_FOR;
    END_FOR;
    
    FOR  k := 0 TO 2 BY 1 DO
        dt_OEE.RecordTime[0,  k].Running     	:= T#0S;
        dt_OEE.RecordTime[0,  k].Stopped     	:= T#0S;
		dt_OEE.RecordTime[0,  k].Error     		:= T#0S;
         
        
         dt_OEE.RecordDate[0]	:=  StartedDate;
         Sts_DailyShiftEnd		:= TRUE;
    END_FOR;
ELSE
     SaveData := FALSE;
END_IF;

IF  dt_OEE.CurrentShift <> 1 THEN
     Sts_DailyShiftEnd := FALSE;
END_IF;

(**Writting Data to Current Shift**)
CASE  dt_OEE.CurrentShift OF
    1:
         dt_OEE.RecordDate[0] :=  StartedDate;
         dt_OEE.RecordTime[0, 0].Running	:=  dt_TimeCal.Running;
         dt_OEE.RecordTime[0, 0].Stopped 	:=  dt_TimeCal.Stopped;
         dt_OEE.RecordTime[0, 0].Error      :=  dt_TimeCal.Error;
    2:
         dt_OEE.RecordDate[0] :=  StartedDate;
         dt_OEE.RecordTime[0, 1].Running 	:=  dt_TimeCal.Running;
         dt_OEE.RecordTime[0, 1].Stopped 	:=  dt_TimeCal.Stopped;
         dt_OEE.RecordTime[0, 1].Error     	:=  dt_TimeCal.Error;
    3:
         dt_OEE.RecordDate[0] :=  StartedDate;
         dt_OEE.RecordTime[0, 2].Running	:=  dt_TimeCal.Running;
         dt_OEE.RecordTime[0, 2].Stopped 	:=  dt_TimeCal.Stopped;
         dt_OEE.RecordTime[0, 2].Error     	:=  dt_TimeCal.Error;
END_CASE;

 dt_OEE.HMI_Date		:=  dt_OEE.RecordDate[ dt_OEE.HMI_NumberPrev];
 dt_OEE.HMI_Time[0] 	:=  dt_OEE.RecordTime[ dt_OEE.HMI_NumberPrev, 0];
 dt_OEE.HMI_Time[1] 	:=  dt_OEE.RecordTime[ dt_OEE.HMI_NumberPrev, 1];
 dt_OEE.HMI_Time[2] 	:=  dt_OEE.RecordTime[ dt_OEE.HMI_NumberPrev, 2];
 
 
 
 dt_OEE.TotalTime.Running		:= dt_OEE.HMI_Time[0].Running + dt_OEE.HMI_Time[1].Running + dt_OEE.HMI_Time[2].Running; 
 dt_OEE.TotalTime.Stopped		:= dt_OEE.HMI_Time[0].Stopped + dt_OEE.HMI_Time[1].Stopped + dt_OEE.HMI_Time[2].Stopped; 
 dt_OEE.TotalTime.Error			:= dt_OEE.HMI_Time[0].Error + dt_OEE.HMI_Time[1].Error + dt_OEE.HMI_Time[2].Error; 

 
 //Elapsed Duration
 IF dt_OEE.CurrentShift = 1 AND dt_OEE.HMI_NumberPrev = 0 THEN
	ShiftDuration[0]			:= TIME_TO_REAL(dt_OEE.TimeCurrent - dt_OEE.TimeShift[1].StartShift);
 ELSE
	ShiftDuration[0]			:= TIME_TO_REAL(T#8H);
 END_IF
 
 IF dt_OEE.CurrentShift = 2 AND dt_OEE.HMI_NumberPrev = 0 THEN
	ShiftDuration[1]			:= TIME_TO_REAL(dt_OEE.TimeCurrent - dt_OEE.TimeShift[2].StartShift);
 ELSE
	ShiftDuration[1]			:= TIME_TO_REAL(T#8H);
 END_IF
 	
 IF dt_OEE.CurrentShift = 3 AND dt_OEE.HMI_NumberPrev = 0 THEN
	 IF dt_OEE.TimeCurrent < dt_OEE.TimeShift[3].EndShift THEN
 		ShiftDuration[2]		:= TOD_TO_REAL(dt_OEE.TimeCurrent + T#2H);
	 ELSE
		ShiftDuration[2]		:= TIME_TO_REAL(dt_OEE.TimeCurrent - dt_OEE.TimeShift[3].StartShift);
	 END_IF
 ELSE
	ShiftDuration[2]			:= TIME_TO_REAL(T#8H);
 END_IF
 
 //Precentage Shift 1
 dt_OEE.Precentage[0].Running		:= (TIME_TO_REAL(dt_OEE.HMI_Time[0].Running)/ShiftDuration[0]) * 100 ;
 dt_OEE.Precentage[0].Stopped		:= (TIME_TO_REAL(dt_OEE.HMI_Time[0].Stopped)/ShiftDuration[0]) * 100 ;
 dt_OEE.Precentage[0].Error			:= (TIME_TO_REAL(dt_OEE.HMI_Time[0].Error)/ShiftDuration[0]) * 100 ;
 //dt_OEE.Precentage[0].Unstated		:= 100 - dt_OEE.Precentage[0].Running - dt_OEE.Precentage[0].Stopped - dt_OEE.Precentage[0].Error;
 
 //Precentage Shift 2
 dt_OEE.Precentage[1].Running		:= (TIME_TO_REAL(dt_OEE.HMI_Time[1].Running)/ShiftDuration[1]) * 100 ;
 dt_OEE.Precentage[1].Stopped		:= (TIME_TO_REAL(dt_OEE.HMI_Time[1].Stopped)/ShiftDuration[1]) * 100 ;
 dt_OEE.Precentage[1].Error			:= (TIME_TO_REAL(dt_OEE.HMI_Time[1].Error)/ShiftDuration[1]) * 100 ;
 //dt_OEE.Precentage[1].Unstated		:= 100 - dt_OEE.Precentage[1].Running - dt_OEE.Precentage[1].Stopped - dt_OEE.Precentage[1].Error;
 
 //Precentage Shift 3
 dt_OEE.Precentage[2].Running		:= (TIME_TO_REAL(dt_OEE.HMI_Time[2].Running)/ShiftDuration[2]) * 100 ;
 dt_OEE.Precentage[2].Stopped		:= (TIME_TO_REAL(dt_OEE.HMI_Time[2].Stopped)/ShiftDuration[2]) * 100 ;
 dt_OEE.Precentage[2].Error			:= (TIME_TO_REAL(dt_OEE.HMI_Time[2].Error)/ShiftDuration[2]) * 100 ;
 //dt_OEE.Precentage[2].Unstated		:= 100 - dt_OEE.Precentage[2].Running - dt_OEE.Precentage[2].Stopped - dt_OEE.Precentage[2].Error;


 //Convert Time To String
 dt_OEE.HMI_Time[0].sRunning	:= ConvertTimeToString(dt_OEE.HMI_Time[0].Running);
 dt_OEE.HMI_Time[0].sStopped	:= ConvertTimeToString(dt_OEE.HMI_Time[0].Stopped);
 dt_OEE.HMI_Time[0].sError		:= ConvertTimeToString(dt_OEE.HMI_Time[0].Error);
 
 dt_OEE.HMI_Time[1].sRunning	:= ConvertTimeToString(dt_OEE.HMI_Time[1].Running);
 dt_OEE.HMI_Time[1].sStopped	:= ConvertTimeToString(dt_OEE.HMI_Time[1].Stopped);
 dt_OEE.HMI_Time[1].sError		:= ConvertTimeToString(dt_OEE.HMI_Time[1].Error);
 
 dt_OEE.HMI_Time[2].sRunning	:= ConvertTimeToString(dt_OEE.HMI_Time[2].Running);
 dt_OEE.HMI_Time[2].sStopped	:= ConvertTimeToString(dt_OEE.HMI_Time[2].Stopped);
 dt_OEE.HMI_Time[2].sError		:= ConvertTimeToString(dt_OEE.HMI_Time[2].Error);
 
IF dt_OEE.HMI_NumberPrev < 0 THEN
	dt_OEE.HMI_NumberPrev := 6;
ELSIF dt_OEE.HMI_NumberPrev > 6  THEN
	dt_OEE.HMI_NumberPrev := 0;
END_IF;

END_FUNCTION_BLOCK

// ---- POUs/Function/ConvertTimeToString.TcPOU
FUNCTION ConvertTimeToString : STRING
VAR_INPUT
	DataInput	: TIME;
END_VAR
VAR
END_VAR

ConvertTimeToString:=DELETE(TOD_TO_STRING(TIME_TO_TOD(DataInput)),5,0);

END_FUNCTION

// ---- POUs/Function_Block/FB_CheckShuttlePos.TcPOU
FUNCTION_BLOCK FB_CheckShuttlePos
VAR_INPUT
	bEnable				: BOOL;
	OFFSET				: DINT;
	ACT					: DINT;
	Shuttle				: ARRAY[0..4] OF stShuttle;
END_VAR
VAR_OUTPUT
	CheckShuttle		: ARRAY [0..4] OF stCheckShuttle;
END_VAR
VAR
	Sequence			: INT;
	DIFF_EMPTY			: DINT;
	DIFF_LOAD			: DINT;
	DIFF_TEMP			: DINT;
	DataTimer			: TON;
	WatchDog			: TON;
	TEMP				: DINT;
	Index				: INT;
	Init				: BOOL;
END_VAR

//Check Postion
IF ABS(TEMP - ACT) > 5 THEN
	DIFF_TEMP := (TEMP - ACT);
ELSE
	DIFF_TEMP := 0;
END_IF;

(* ================== Check Shuttle Position ================== *)
IF (DIFF_TEMP <> 0 AND ACT <> 0) OR NOT Init THEN
	FOR Index := 0 TO 4 BY 1 DO
		//Check Empty Pallet Position
		IF ABS(Shuttle[Index].PositionEmpty - ACT) > OFFSET THEN
			DIFF_EMPTY := (Shuttle[Index].PositionEmpty - ACT);
		ELSE
			DIFF_EMPTY := 0;
		END_IF;
		
		IF DIFF_EMPTY = 0 THEN
			CheckShuttle[Index].AtEmpty := TRUE;
		ELSE
			CheckShuttle[Index].AtEmpty := FALSE;
		END_IF 	
		
		//Check Load Pallet Position
		IF ABS(Shuttle[Index].PositionLoaded - ACT) > OFFSET THEN
			DIFF_LOAD := (Shuttle[Index].PositionLoaded - ACT);
		ELSE
			DIFF_LOAD := 0;
		END_IF;
		
		IF DIFF_LOAD = 0 THEN
			CheckShuttle[Index].AtLoad := TRUE;
		ELSE
			CheckShuttle[Index].AtLoad := FALSE;
		END_IF 	
	
	END_FOR
	//Update Position
	TEMP	:= ACT;	
	Init	:= TRUE;
END_IF

END_FUNCTION_BLOCK

// ---- POUs/Function_Block/General/OEECounter.TcPOU
FUNCTION_BLOCK OEECounter
VAR_INPUT
	ENI					: BOOL;
	CurrentTime			: DT;
	dt_Production		: ShiftCounter;
END_VAR
VAR_OUTPUT 
	bGetData			: BOOL;
END_VAR
VAR_IN_OUT PERSISTENT
	dt_OEE				: sOEECounter;
END_VAR
VAR PERSISTENT
	StartedDate			: DATE;
	StartedShift		: UINT;
	Sts_DailyShiftEnd	: BOOL;
	SaveData			: BOOL;
	i					: INT;
	j					: INT;
	k					: INT;
	l					: INT;
	m					: INT;
	n					: INT;
END_VAR

//Get Time & Parsing
dt_OEE.DateCurrent := DT_TO_DATE(CurrentTime);
dt_OEE.TimeCurrent := DT_TO_TOD(CurrentTime);

dt_OEE.TimeShift[1].StartShift	:= TOD#06:00:00;
dt_OEE.TimeShift[2].StartShift	:= TOD#14:00:00;
dt_OEE.TimeShift[3].StartShift	:= TOD#22:00:00;

dt_OEE.TimeShift[1].EndShift	:= TOD#14:00:00;
dt_OEE.TimeShift[2].EndShift	:= TOD#22:00:00;
dt_OEE.TimeShift[3].EndShift	:= TOD#06:00:00;

(**Get Data**)
IF (( dt_OEE.TimeCurrent >  dt_OEE.TimeShift[1].EndShift) AND ( dt_OEE.TimeCurrent < dt_OEE.TimeShift[1].EndShift + T#3S)) 
    OR (( dt_OEE.TimeCurrent >  dt_OEE.TimeShift[2].EndShift) AND ( dt_OEE.TimeCurrent < dt_OEE.TimeShift[2].EndShift + T#3S)) 
    OR (( dt_OEE.TimeCurrent >  dt_OEE.TimeShift[3].EndShift) AND ( dt_OEE.TimeCurrent < dt_OEE.TimeShift[3].EndShift + T#3S))  THEN
    IF NOT  bGetData THEN
         bGetData := TRUE;
         StartedDate	:=  dt_OEE.DateCurrent;
         StartedShift	:=  dt_OEE.CurrentShift;
    END_IF;
ELSE
     bGetData := FALSE;
END_IF;

(**Shift Checking**)
IF NOT  SaveData THEN
    IF ( dt_OEE.TimeCurrent >  dt_OEE.TimeShift[1].StartShift) AND ( dt_OEE.TimeCurrent <  dt_OEE.TimeShift[1].EndShift) THEN
         dt_OEE.CurrentShift := 1;
    ELSIF ( dt_OEE.TimeCurrent >  dt_OEE.TimeShift[2].StartShift) AND ( dt_OEE.TimeCurrent <  dt_OEE.TimeShift[2].EndShift) THEN
         dt_OEE.CurrentShift := 2;
    ELSIF ( dt_OEE.TimeCurrent >  dt_OEE.TimeShift[3].StartShift) OR ( dt_OEE.TimeCurrent <  dt_OEE.TimeShift[3].EndShift) THEN
         dt_OEE.CurrentShift := 3;
    END_IF;
END_IF;

(** Function to Clear Data Record **)
(*IF dt_OEE.Reset THEN	
	    FOR m := 1 TO 6 BY 1 DO
	        FOR n := 0 TO 2 BY 1 DO
	            dt_OEE.CounterRecord[m, n].Data1 		:= 0;
	            dt_OEE.CounterRecord[m, n].Data2		:= 0;
	            dt_OEE.CounterRecord[m, n].Data3 		:= 0;
	            dt_OEE.CounterRecord[m, n].Data4 		:= 0;
				dt_OEE.CounterRecord[m, n].ProductCode 	:='';
	        END_FOR;
	    END_FOR;
END_IF;*)

(** Function to copy daily information to history AND Reset Timer**)
IF (( dt_OEE.TimeCurrent >  dt_OEE.TimeShift[3].EndShift) AND ( dt_OEE.TimeCurrent < ( dt_OEE.TimeShift[3].EndShift+T#3S))) AND NOT Sts_DailyShiftEnd THEN
    SaveData := TRUE;
	    FOR j := 5 TO 0 BY -1 DO
	        FOR k := 0 TO 2 BY 1 DO
	            dt_OEE.CounterRecord[j + 1, k].Data1 		:= dt_OEE.CounterRecord[j, k].Data1;
	            dt_OEE.CounterRecord[j + 1, k].Data2 		:= dt_OEE.CounterRecord[j, k].Data2;
	            dt_OEE.CounterRecord[j + 1, k].Data3 		:= dt_OEE.CounterRecord[j, k].Data3;
	            dt_OEE.CounterRecord[j + 1, k].Data4 		:= dt_OEE.CounterRecord[j, k].Data4;
				dt_OEE.CounterRecord[j + 1, k].ProductCode 	:= dt_OEE.CounterRecord[j, k].ProductCode;
	            dt_OEE.DateRecord[j + 1] 					:= dt_OEE.DateRecord[j];
	        END_FOR;
	    END_FOR;
		
	    FOR l := 0 TO 2 BY 1 DO
	        dt_OEE.CounterRecord[0, l].Data1 		:= 0;
	        dt_OEE.CounterRecord[0, l].Data2 		:= 0;
	        dt_OEE.CounterRecord[0, l].Data3 		:= 0;
	        dt_OEE.CounterRecord[0, l].Data4 		:= 0;
			dt_OEE.CounterRecord[0, l].ProductCode 		:='';
	        Sts_DailyShiftEnd := TRUE;
	    END_FOR;
ELSE
    SaveData := FALSE;
END_IF;

IF dt_OEE.CurrentShift <> 1 THEN
    Sts_DailyShiftEnd := FALSE;
END_IF;

CASE t_OEE.CurrentShift OF
	1:
		dt_OEE.DateRecord[0] := StartedDate;
		dt_OEE.CounterRecord[ 0,0].ProductCode := Dt_Production.ProductCode;
		dt_OEE.CounterRecord[ 0,0].Data1 := Dt_Production.Data1;
		dt_OEE.CounterRecord[ 0,0].Data2 := Dt_Production.Data2;
		dt_OEE.CounterRecord[ 0,0].Data3 := Dt_Production.Data3;
	2:
		dt_OEE.CounterRecord[ 0,1].ProductCode := Dt_Production.ProductCode;
		dt_OEE.CounterRecord[ 0,1].Data1 := Dt_Production.Data1;
		dt_OEE.CounterRecord[ 0,1].Data2 := Dt_Production.Data2;
		dt_OEE.CounterRecord[ 0,1].Data3 := Dt_Production.Data3;
	3:
		dt_OEE.CounterRecord[ 0,2].ProductCode := Dt_Production.ProductCode;
		dt_OEE.CounterRecord[ 0,2].Data1 := Dt_Production.Data1;
		dt_OEE.CounterRecord[ 0,2].Data2 := Dt_Production.Data2;
		dt_OEE.CounterRecord[ 0,2].Data3 := Dt_Production.Data3;
END_CASE;

(**Writting Data to Current Shift**)
//======================== Line ========================//

dt_OEE.HMI_Counter[0] := dt_OEE.CounterRecord[Dt_OEE.HMI_NumberPrev,0];
dt_OEE.HMI_Counter[1] := dt_OEE.CounterRecord[Dt_OEE.HMI_NumberPrev,1];
dt_OEE.HMI_Counter[2] := dt_OEE.CounterRecord[Dt_OEE.HMI_NumberPrev,2];

//Total Counter
Dt_OEE.TotalCounter.Data1	:= dt_OEE.HMI_Counter[0].Data1 + dt_OEE.HMI_Counter[1].Data1 + dt_OEE.HMI_Counter[2].Data1;
Dt_OEE.TotalCounter.Data2	:= dt_OEE.HMI_Counter[0].Data2 + dt_OEE.HMI_Counter[1].Data2 + dt_OEE.HMI_Counter[2].Data2;
Dt_OEE.TotalCounter.Data3	:= dt_OEE.HMI_Counter[0].Data3 + dt_OEE.HMI_Counter[1].Data3 + dt_OEE.HMI_Counter[2].Data3;
Dt_OEE.TotalCounter.Data4	:= dt_OEE.HMI_Counter[0].Data4 + dt_OEE.HMI_Counter[1].Data4 + dt_OEE.HMI_Counter[2].Data4;

 
IF dt_OEE.HMI_NumberPrev < 0 THEN
	dt_OEE.HMI_NumberPrev := 6;
ELSIF dt_OEE.HMI_NumberPrev > 6  THEN
	dt_OEE.HMI_NumberPrev := 0;
END_IF;

END_FUNCTION_BLOCK

// ---- POUs/S01_Robot/EM01_Robot.TcPOU
PROGRAM EM01_Robot
VAR
	
	//Backbone
	FB_StateMachine_Robot			: FB_StateManager;
	bFl_RunningMachineRobot			: BOOL;
	bFl_SeqReset					: BOOL;
	Bypass_Safety					: BOOL;
	bFl_Manual						: BOOL;
	CheckStatusRobot				: checkstatus;
	AlarmEventHistory				: ARRAY[1..20] OF Alarm_Event_History;
	StartUpRobot					: FB_StartUpRobot;
	AlarmEventActive				: ARRAY[1..20] OF Alarm_Event_Active;
	Connection_Robot				: TON;
END_VAR
VAR // added by the converter: edge detectors and wires of the graphical bodies
    _w1, _w2, _w3, _w4 : BOOL;
END_VAR

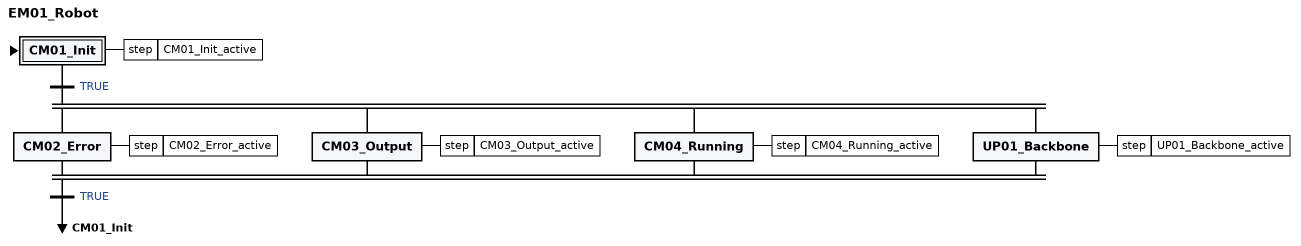
INITIAL_STEP CM01_Init:
    CM01_Init_active(N);  // step action
END_STEP
TRANSITION FROM CM01_Init TO (CM02_Error, CM03_Output, CM04_Running, UP01_Backbone)
    := TRUE;
END_TRANSITION
STEP CM02_Error:
    CM02_Error_active(N);  // step action
END_STEP
STEP CM03_Output:
    CM03_Output_active(N);  // step action
END_STEP
STEP CM04_Running:
    CM04_Running_active(N);  // step action
END_STEP
STEP UP01_Backbone:
    UP01_Backbone_active(N);  // step action
END_STEP
TRANSITION FROM (CM02_Error, CM03_Output, CM04_Running, UP01_Backbone) TO CM01_Init
    := TRUE;
END_TRANSITION

ACTION CM01_Init_active:
Data_GVL.bFL_StartRobot				:= Status_GVL.bFl_RunButton_Robotic OR HMI_GVL.bStartButtonRobot;
Data_GVL.bFL_StopRobot				:= NOT Status_GVL.bFl_StopButton_Robotic OR HMI_GVL.bStopButtonRobot;
Data_GVL.bFL_ResetRobot				:= Status_GVL.bFl_ResetButton_Robotic OR HMI_GVL.bResetButtonRobot;
Data_GVL.bFL_AckRobot				:= Status_GVL.bFl_Acknowledge_Robotic OR HMI_GVL.bAcknowledgeButtonRobot;
Data_GVL.bFL_AutoManuaModeRobot 	:= Status_GVL.bFl_Manual_Robotic OR HMI_GVL.bTestModeEnableRobot;
bFl_RunningMachineRobot				:= Data_GVL.stStateMachineRobot.Running;
bFl_Manual							:= Data_GVL.stStateMachineRobot.ManualMode;
bFl_SeqReset						:= NOT Status_GVL.bFl_EStop_Robotic OR InputOutput_GVL.xIn_Robot.StsSupervision OR InputOutput_GVL.xIn_Robot.StsEmergencyStop OR NOT InputOutput_GVL.xIn_Robot.StsAutoOn;



(*=================Convert Timer============================*)
END_ACTION

ACTION CM02_Error_active:
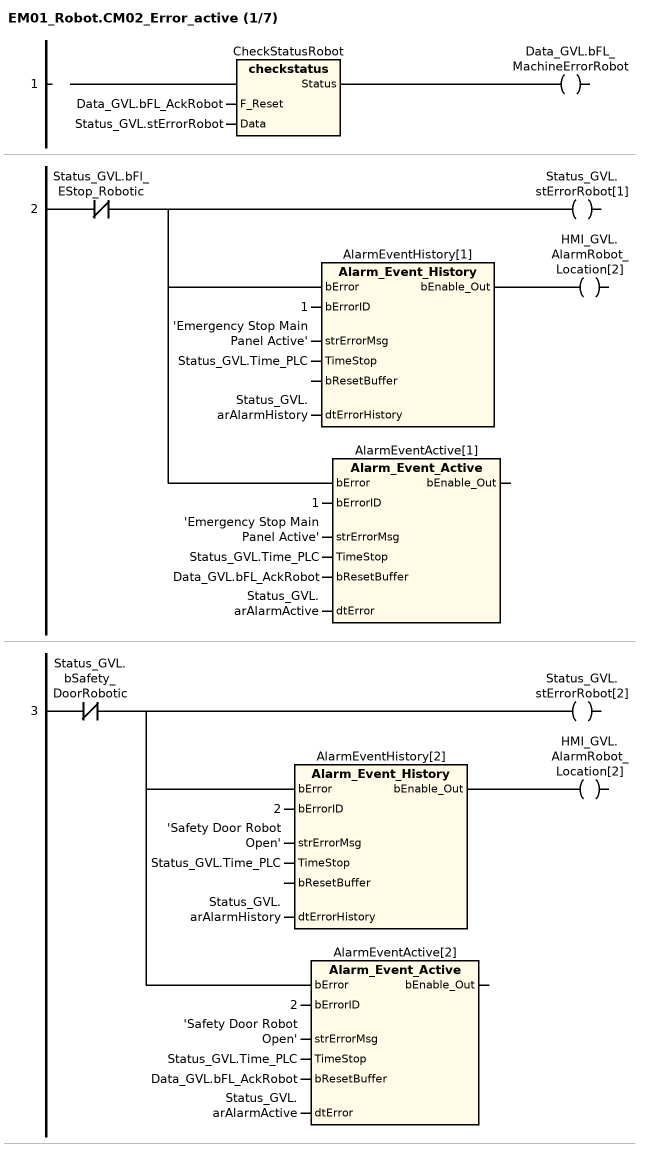
// NETWORK 1
CheckStatusRobot(F_Reset := Data_GVL.bFL_AckRobot, Data := Status_GVL.stErrorRobot); // checkstatus
Data_GVL.bFL_MachineErrorRobot := CheckStatusRobot.Status;

// NETWORK 2
_w1 := NOT Status_GVL.bFl_EStop_Robotic;
Status_GVL.stErrorRobot[1] := _w1;
AlarmEventHistory[1](
    bError := _w1,
    bErrorID := 1,
    strErrorMsg := 'Emergency Stop Main Panel Active',
    TimeStop := Status_GVL.Time_PLC,
    dtErrorHistory := Status_GVL.arAlarmHistory); // Alarm_Event_History
HMI_GVL.AlarmRobot_Location[2] := AlarmEventHistory[1].bEnable_Out;
AlarmEventActive[1](
    bError := _w1,
    bErrorID := 1,
    strErrorMsg := 'Emergency Stop Main Panel Active',
    TimeStop := Status_GVL.Time_PLC,
    bResetBuffer := Data_GVL.bFL_AckRobot,
    dtError := Status_GVL.arAlarmActive); // Alarm_Event_Active

// NETWORK 3
_w2 := NOT Status_GVL.bSafety_DoorRobotic;
Status_GVL.stErrorRobot[2] := _w2;
AlarmEventHistory[2](
    bError := _w2,
    bErrorID := 2,
    strErrorMsg := 'Safety Door Robot Open',
    TimeStop := Status_GVL.Time_PLC,
    dtErrorHistory := Status_GVL.arAlarmHistory); // Alarm_Event_History
HMI_GVL.AlarmRobot_Location[2] := AlarmEventHistory[2].bEnable_Out;
AlarmEventActive[2](
    bError := _w2,
    bErrorID := 2,
    strErrorMsg := 'Safety Door Robot Open',
    TimeStop := Status_GVL.Time_PLC,
    bResetBuffer := Data_GVL.bFL_AckRobot,
    dtError := Status_GVL.arAlarmActive); // Alarm_Event_Active

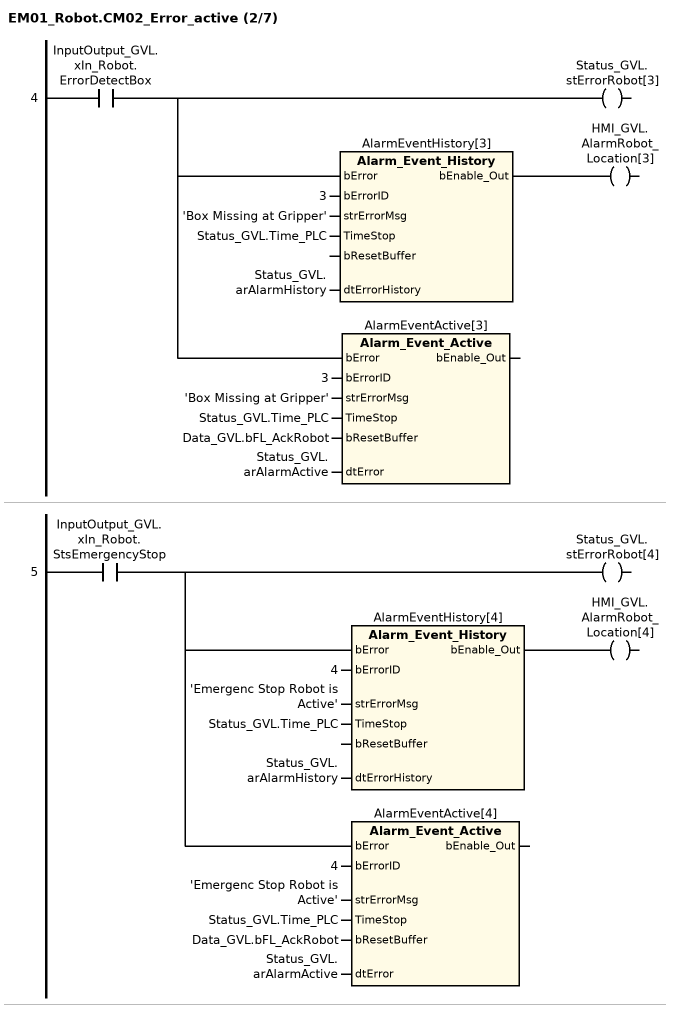
// NETWORK 4
Status_GVL.stErrorRobot[3] := InputOutput_GVL.xIn_Robot.ErrorDetectBox;
AlarmEventHistory[3](
    bError := InputOutput_GVL.xIn_Robot.ErrorDetectBox,
    bErrorID := 3,
    strErrorMsg := 'Box Missing at Gripper',
    TimeStop := Status_GVL.Time_PLC,
    dtErrorHistory := Status_GVL.arAlarmHistory); // Alarm_Event_History
HMI_GVL.AlarmRobot_Location[3] := AlarmEventHistory[3].bEnable_Out;
AlarmEventActive[3](
    bError := InputOutput_GVL.xIn_Robot.ErrorDetectBox,
    bErrorID := 3,
    strErrorMsg := 'Box Missing at Gripper',
    TimeStop := Status_GVL.Time_PLC,
    bResetBuffer := Data_GVL.bFL_AckRobot,
    dtError := Status_GVL.arAlarmActive); // Alarm_Event_Active

// NETWORK 5
Status_GVL.stErrorRobot[4] := InputOutput_GVL.xIn_Robot.StsEmergencyStop;
AlarmEventHistory[4](
    bError := InputOutput_GVL.xIn_Robot.StsEmergencyStop,
    bErrorID := 4,
    strErrorMsg := 'Emergenc Stop Robot is Active',
    TimeStop := Status_GVL.Time_PLC,
    dtErrorHistory := Status_GVL.arAlarmHistory); // Alarm_Event_History
HMI_GVL.AlarmRobot_Location[4] := AlarmEventHistory[4].bEnable_Out;
AlarmEventActive[4](
    bError := InputOutput_GVL.xIn_Robot.StsEmergencyStop,
    bErrorID := 4,
    strErrorMsg := 'Emergenc Stop Robot is Active',
    TimeStop := Status_GVL.Time_PLC,
    bResetBuffer := Data_GVL.bFL_AckRobot,
    dtError := Status_GVL.arAlarmActive); // Alarm_Event_Active

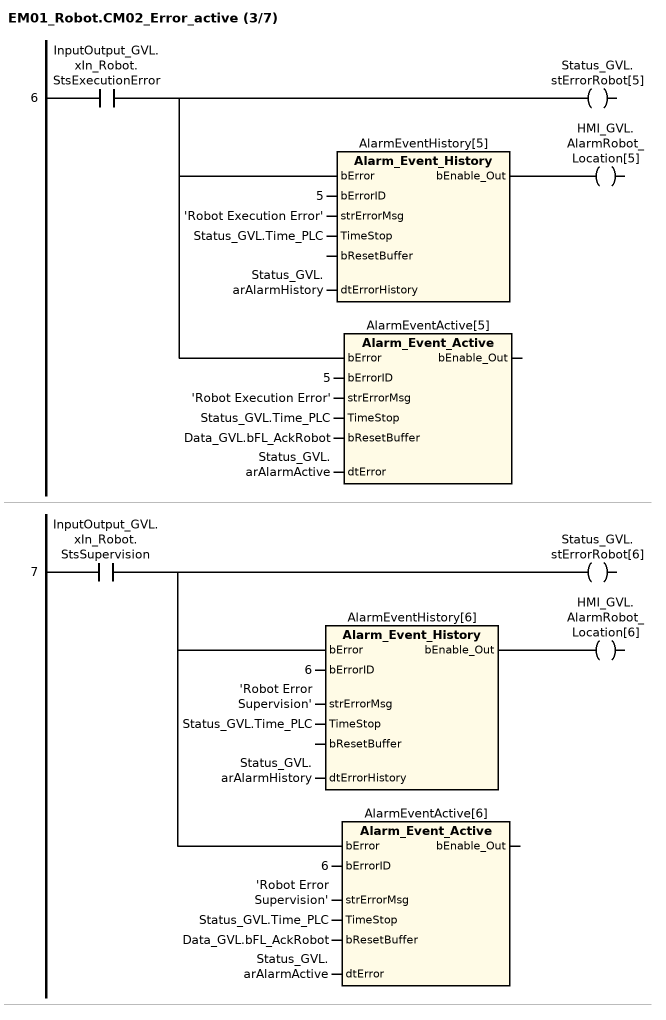
// NETWORK 6
Status_GVL.stErrorRobot[5] := InputOutput_GVL.xIn_Robot.StsExecutionError;
AlarmEventHistory[5](
    bError := InputOutput_GVL.xIn_Robot.StsExecutionError,
    bErrorID := 5,
    strErrorMsg := 'Robot Execution Error',
    TimeStop := Status_GVL.Time_PLC,
    dtErrorHistory := Status_GVL.arAlarmHistory); // Alarm_Event_History
HMI_GVL.AlarmRobot_Location[5] := AlarmEventHistory[5].bEnable_Out;
AlarmEventActive[5](
    bError := InputOutput_GVL.xIn_Robot.StsExecutionError,
    bErrorID := 5,
    strErrorMsg := 'Robot Execution Error',
    TimeStop := Status_GVL.Time_PLC,
    bResetBuffer := Data_GVL.bFL_AckRobot,
    dtError := Status_GVL.arAlarmActive); // Alarm_Event_Active

// NETWORK 7
Status_GVL.stErrorRobot[6] := InputOutput_GVL.xIn_Robot.StsSupervision;
AlarmEventHistory[6](
    bError := InputOutput_GVL.xIn_Robot.StsSupervision,
    bErrorID := 6,
    strErrorMsg := 'Robot Error Supervision',
    TimeStop := Status_GVL.Time_PLC,
    dtErrorHistory := Status_GVL.arAlarmHistory); // Alarm_Event_History
HMI_GVL.AlarmRobot_Location[6] := AlarmEventHistory[6].bEnable_Out;
AlarmEventActive[6](
    bError := InputOutput_GVL.xIn_Robot.StsSupervision,
    bErrorID := 6,
    strErrorMsg := 'Robot Error Supervision',
    TimeStop := Status_GVL.Time_PLC,
    bResetBuffer := Data_GVL.bFL_AckRobot,
    dtError := Status_GVL.arAlarmActive); // Alarm_Event_Active

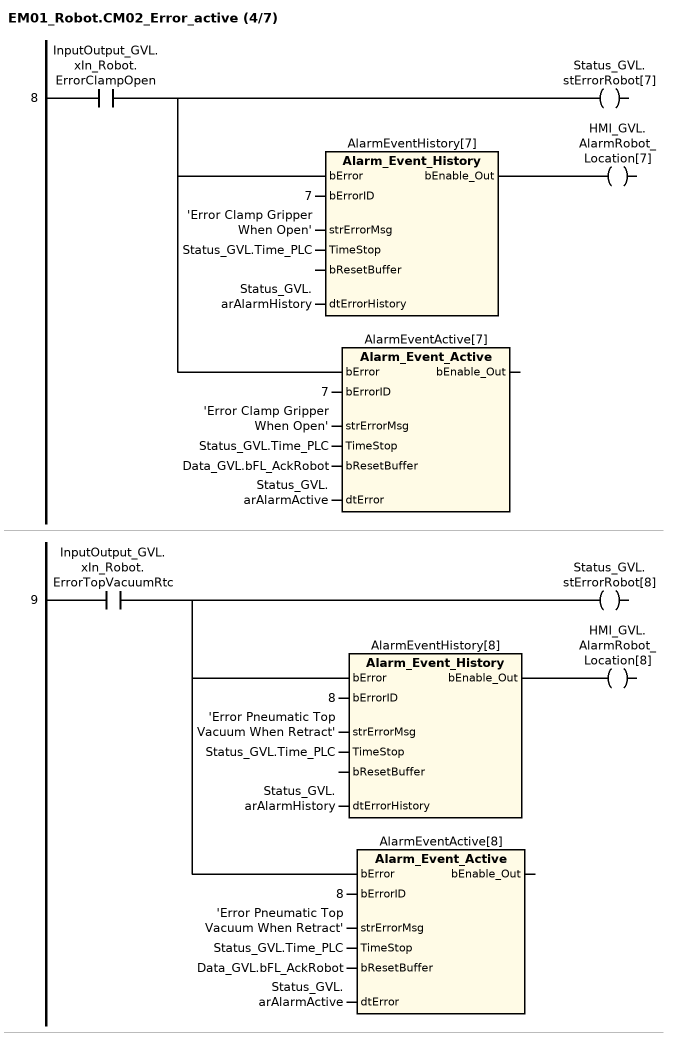
// NETWORK 8
Status_GVL.stErrorRobot[7] := InputOutput_GVL.xIn_Robot.ErrorClampOpen;
AlarmEventHistory[7](
    bError := InputOutput_GVL.xIn_Robot.ErrorClampOpen,
    bErrorID := 7,
    strErrorMsg := 'Error Clamp Gripper When Open',
    TimeStop := Status_GVL.Time_PLC,
    dtErrorHistory := Status_GVL.arAlarmHistory); // Alarm_Event_History
HMI_GVL.AlarmRobot_Location[7] := AlarmEventHistory[7].bEnable_Out;
AlarmEventActive[7](
    bError := InputOutput_GVL.xIn_Robot.ErrorClampOpen,
    bErrorID := 7,
    strErrorMsg := 'Error Clamp Gripper When Open',
    TimeStop := Status_GVL.Time_PLC,
    bResetBuffer := Data_GVL.bFL_AckRobot,
    dtError := Status_GVL.arAlarmActive); // Alarm_Event_Active

// NETWORK 9
Status_GVL.stErrorRobot[8] := InputOutput_GVL.xIn_Robot.ErrorTopVacuumRtc;
AlarmEventHistory[8](
    bError := InputOutput_GVL.xIn_Robot.ErrorTopVacuumRtc,
    bErrorID := 8,
    strErrorMsg := 'Error Pneumatic Top Vacuum When Retract',
    TimeStop := Status_GVL.Time_PLC,
    dtErrorHistory := Status_GVL.arAlarmHistory); // Alarm_Event_History
HMI_GVL.AlarmRobot_Location[8] := AlarmEventHistory[8].bEnable_Out;
AlarmEventActive[8](
    bError := InputOutput_GVL.xIn_Robot.ErrorTopVacuumRtc,
    bErrorID := 8,
    strErrorMsg := 'Error Pneumatic Top Vacuum When Retract',
    TimeStop := Status_GVL.Time_PLC,
    bResetBuffer := Data_GVL.bFL_AckRobot,
    dtError := Status_GVL.arAlarmActive); // Alarm_Event_Active

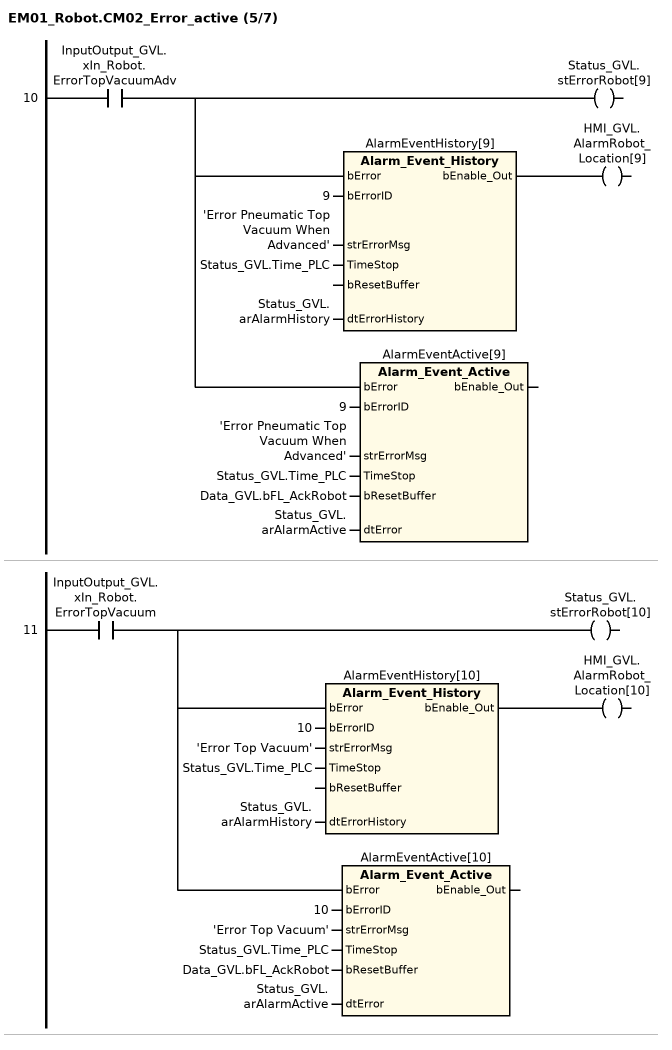
// NETWORK 10
Status_GVL.stErrorRobot[9] := InputOutput_GVL.xIn_Robot.ErrorTopVacuumAdv;
AlarmEventHistory[9](
    bError := InputOutput_GVL.xIn_Robot.ErrorTopVacuumAdv,
    bErrorID := 9,
    strErrorMsg := 'Error Pneumatic Top Vacuum When Advanced',
    TimeStop := Status_GVL.Time_PLC,
    dtErrorHistory := Status_GVL.arAlarmHistory); // Alarm_Event_History
HMI_GVL.AlarmRobot_Location[9] := AlarmEventHistory[9].bEnable_Out;
AlarmEventActive[9](
    bError := InputOutput_GVL.xIn_Robot.ErrorTopVacuumAdv,
    bErrorID := 9,
    strErrorMsg := 'Error Pneumatic Top Vacuum When Advanced',
    TimeStop := Status_GVL.Time_PLC,
    bResetBuffer := Data_GVL.bFL_AckRobot,
    dtError := Status_GVL.arAlarmActive); // Alarm_Event_Active

// NETWORK 11
Status_GVL.stErrorRobot[10] := InputOutput_GVL.xIn_Robot.ErrorTopVacuum;
AlarmEventHistory[10](
    bError := InputOutput_GVL.xIn_Robot.ErrorTopVacuum,
    bErrorID := 10,
    strErrorMsg := 'Error Top Vacuum',
    TimeStop := Status_GVL.Time_PLC,
    dtErrorHistory := Status_GVL.arAlarmHistory); // Alarm_Event_History
HMI_GVL.AlarmRobot_Location[10] := AlarmEventHistory[10].bEnable_Out;
AlarmEventActive[10](
    bError := InputOutput_GVL.xIn_Robot.ErrorTopVacuum,
    bErrorID := 10,
    strErrorMsg := 'Error Top Vacuum',
    TimeStop := Status_GVL.Time_PLC,
    bResetBuffer := Data_GVL.bFL_AckRobot,
    dtError := Status_GVL.arAlarmActive); // Alarm_Event_Active

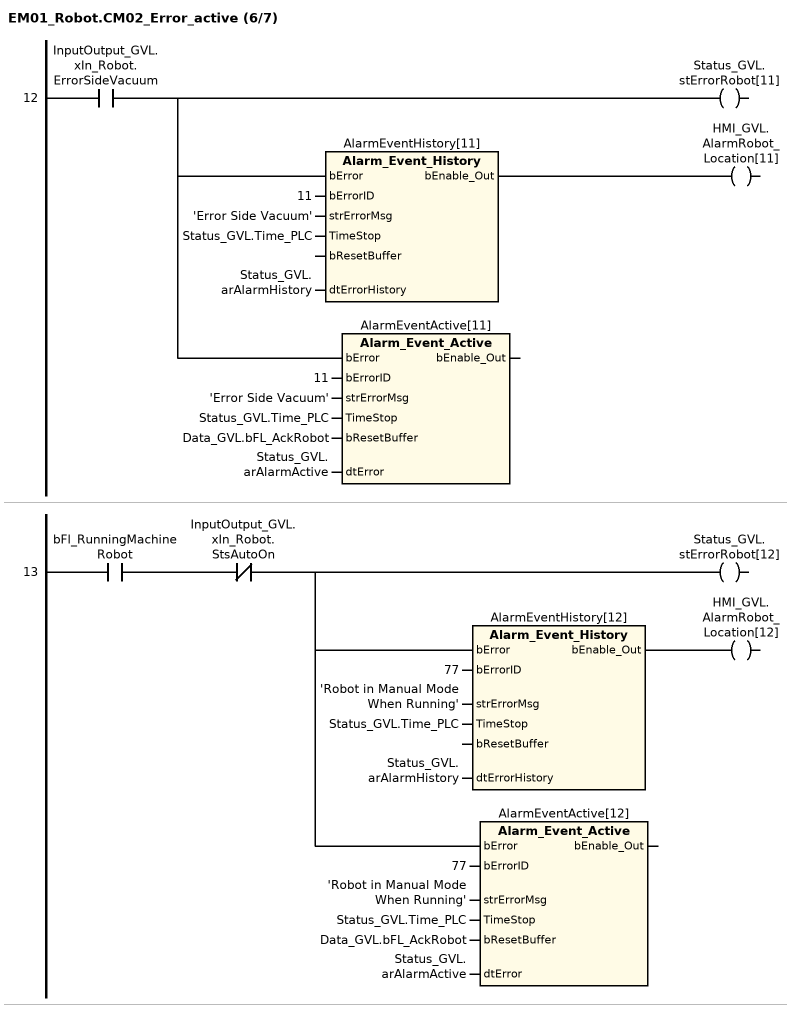
// NETWORK 12
Status_GVL.stErrorRobot[11] := InputOutput_GVL.xIn_Robot.ErrorSideVacuum;
AlarmEventHistory[11](
    bError := InputOutput_GVL.xIn_Robot.ErrorSideVacuum,
    bErrorID := 11,
    strErrorMsg := 'Error Side Vacuum',
    TimeStop := Status_GVL.Time_PLC,
    dtErrorHistory := Status_GVL.arAlarmHistory); // Alarm_Event_History
HMI_GVL.AlarmRobot_Location[11] := AlarmEventHistory[11].bEnable_Out;
AlarmEventActive[11](
    bError := InputOutput_GVL.xIn_Robot.ErrorSideVacuum,
    bErrorID := 11,
    strErrorMsg := 'Error Side Vacuum',
    TimeStop := Status_GVL.Time_PLC,
    bResetBuffer := Data_GVL.bFL_AckRobot,
    dtError := Status_GVL.arAlarmActive); // Alarm_Event_Active

// NETWORK 13
_w3 := bFl_RunningMachineRobot AND NOT InputOutput_GVL.xIn_Robot.StsAutoOn;
Status_GVL.stErrorRobot[12] := _w3;
AlarmEventHistory[12](
    bError := _w3,
    bErrorID := 77,
    strErrorMsg := 'Robot in Manual Mode When Running',
    TimeStop := Status_GVL.Time_PLC,
    dtErrorHistory := Status_GVL.arAlarmHistory); // Alarm_Event_History
HMI_GVL.AlarmRobot_Location[12] := AlarmEventHistory[12].bEnable_Out;
AlarmEventActive[12](
    bError := _w3,
    bErrorID := 77,
    strErrorMsg := 'Robot in Manual Mode When Running',
    TimeStop := Status_GVL.Time_PLC,
    bResetBuffer := Data_GVL.bFL_AckRobot,
    dtError := Status_GVL.arAlarmActive); // Alarm_Event_Active

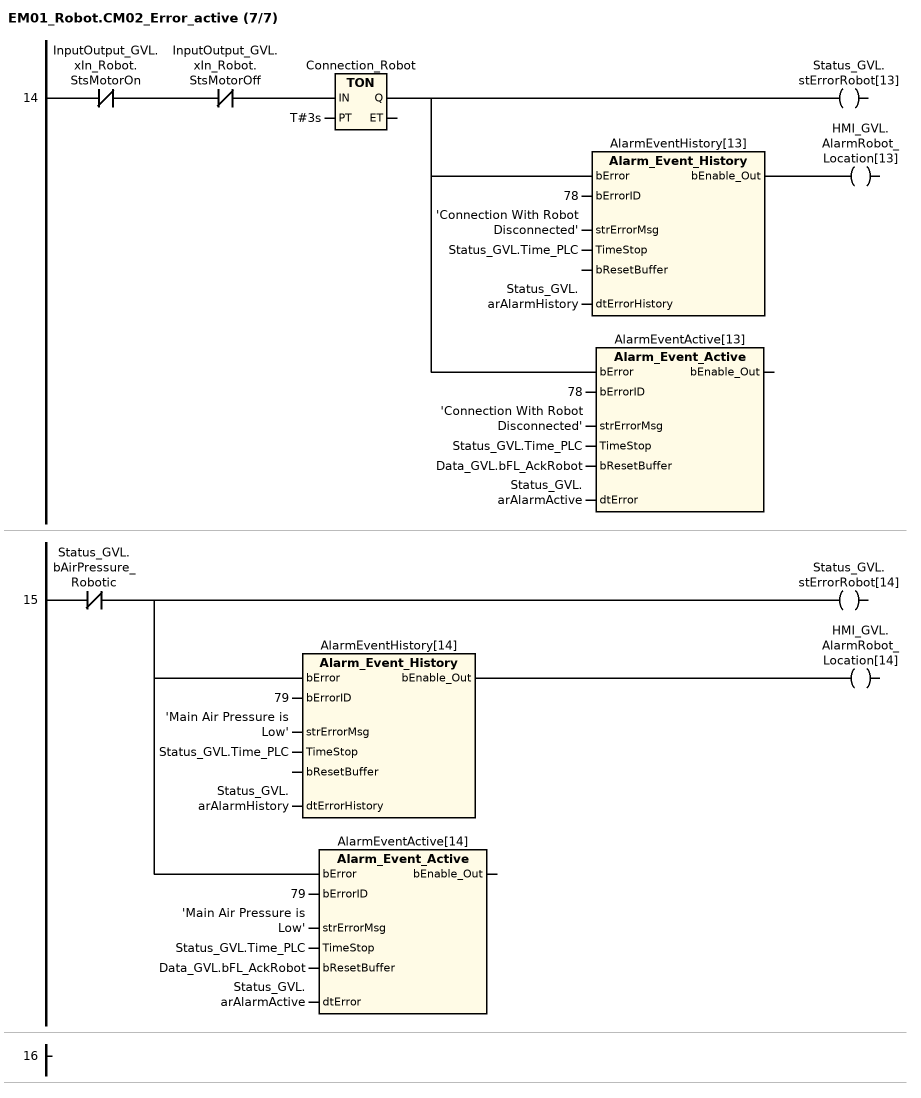
// NETWORK 14
Connection_Robot(IN := NOT InputOutput_GVL.xIn_Robot.StsMotorOn AND NOT InputOutput_GVL.xIn_Robot.StsMotorOff, PT := T#3s); // TON
Status_GVL.stErrorRobot[13] := Connection_Robot.Q;
AlarmEventHistory[13](
    bError := Connection_Robot.Q,
    bErrorID := 78,
    strErrorMsg := 'Connection With Robot Disconnected',
    TimeStop := Status_GVL.Time_PLC,
    dtErrorHistory := Status_GVL.arAlarmHistory); // Alarm_Event_History
HMI_GVL.AlarmRobot_Location[13] := AlarmEventHistory[13].bEnable_Out;
AlarmEventActive[13](
    bError := Connection_Robot.Q,
    bErrorID := 78,
    strErrorMsg := 'Connection With Robot Disconnected',
    TimeStop := Status_GVL.Time_PLC,
    bResetBuffer := Data_GVL.bFL_AckRobot,
    dtError := Status_GVL.arAlarmActive); // Alarm_Event_Active

// NETWORK 15
_w4 := NOT Status_GVL.bAirPressure_Robotic;
Status_GVL.stErrorRobot[14] := _w4;
AlarmEventHistory[14](
    bError := _w4,
    bErrorID := 79,
    strErrorMsg := 'Main Air Pressure is Low',
    TimeStop := Status_GVL.Time_PLC,
    dtErrorHistory := Status_GVL.arAlarmHistory); // Alarm_Event_History
HMI_GVL.AlarmRobot_Location[14] := AlarmEventHistory[14].bEnable_Out;
AlarmEventActive[14](
    bError := _w4,
    bErrorID := 79,
    strErrorMsg := 'Main Air Pressure is Low',
    TimeStop := Status_GVL.Time_PLC,
    bResetBuffer := Data_GVL.bFL_AckRobot,
    dtError := Status_GVL.arAlarmActive); // Alarm_Event_Active

// NETWORK 16
END_ACTION

ACTION CM03_Output_active:
// NETWORK 1 (disabled)
// label: Output Robot
END_ACTION

ACTION CM04_Running_active:
